(* --- decide -------------------------------------------------------------------
   An end stop is driven into rather than stopped at: the motor keeps running for
   T_EndStop once the estimate reaches the limit, which is what makes the position
   measured there rather than integrated forever, and what lets a cover that has
   drifted find itself again. *)
(* --- a full command re-references, and does not trust the estimate ------------
   The run is timed from the whole travel time rather than from the distance the
   estimate believes is left. That distinction is the difference between a cover
   that heals and one that cannot: if the estimate reads 80 while the shutter is
   at 20, a run of "the remaining 20%" ends nowhere near the stop and the error
   survives. A run of the full travel always ends against it.

   The timer only accumulates while a motor is actually turning, so a fbLockout
   delay or a PRIO_LOCK pause does not eat into the travel - and a lock that
   interrupts a run restarts it from the beginning, which is the safe direction to
   fail in. *)
IF rTarget >= 100.0 THEN
	tRefTime := T_TravelUp + T_EndStop;
ELSE
	tRefTime := T_TravelDown + T_EndStop;
END_IF

fbRefRun(IN := bReferencing AND (iDrivingLast <> ciDriveStop), PT := tRefTime);

IF iManualDrive <> ciDriveStop THEN
	iDriving := iManualDrive;

ELSIF bArrived THEN
	(* Nothing outstanding. Without this the motor restarts the moment a timer
	   resets, and the cover hunts at the limit forever. *)
	iDriving := ciDriveStop;

ELSIF bReferencing THEN
	IF fbRefRun.Q THEN
		(* Against the stop by the clock. This is the one moment the position is
		   measured rather than integrated, so the estimate is set, not nudged. *)
		iDriving := ciDriveStop;
		bArrived := TRUE;
		bReferencing := FALSE;
		PositionKnown := TRUE;
		IF rTarget >= 100.0 THEN
			rPositionReal := 100.0;
		ELSE
			rPositionReal := 0.0;
		END_IF
	ELSIF rTarget >= 100.0 THEN
		iDriving := ciDriveUp;
	ELSE
		iDriving := ciDriveDown;
	END_IF

ELSIF (rTarget - rPositionReal) > BYTE_TO_REAL(Tolerance) THEN
	iDriving := ciDriveUp;

ELSIF (rPositionReal - rTarget) > BYTE_TO_REAL(Tolerance) THEN
	iDriving := ciDriveDown;

ELSE
	(* Close enough. A shutter cannot be positioned finer than its own start and
	   stop time, so this is where a mid-range journey ends - and a mid-range
	   journey is the one case that cannot re-reference, because it does not go
	   anywhere the position is known. *)
	iDriving := ciDriveStop;
	bArrived := TRUE;
END_IF

IF PRIO_LOCK THEN
	iDriving := ciDriveStop;
END_IF

(* --- fbLockout ------------------------------------------------------------------
   A reversing contactor must never be asked to change direction while the motor
   is still turning, so a direction change always passes through a stop of at
   least T_Lockout. Starting from standstill is not delayed. *)
IF (iDriving <> ciDriveStop) AND (iDrivingLast <> ciDriveStop) AND (iDriving <> iDrivingLast) THEN
	iDriving := ciDriveStop;
END_IF

(* The timer runs on where the cover WAS, not on what has just been decided.
   Feeding it the decision deadlocks the block: asking to move makes IN FALSE,
   which resets the very timer that would have permitted moving, so the request
   is refused again on the next cycle and forever after. That cost a bench run,
   and the symptom was a cover that byReported STOPPED at 0% no matter what was
   asked of it. *)
fbLockout(IN := (iDrivingLast = ciDriveStop), PT := T_Lockout);

IF (iDriving <> ciDriveStop) AND (iDrivingLast = ciDriveStop) AND NOT fbLockout.Q THEN
	(* Stopped too recently to start again - the contactor gets its dead time. *)
	iDriving := ciDriveStop;
END_IF

iDrivingLast := iDriving;

MU := (iDriving = ciDriveUp);
MD := (iDriving = ciDriveDown);
Moving := MU OR MD;
Position := REAL_TO_BYTE(rPositionReal + 0.5);

(* --- what to tell Home Assistant ---------------------------------------------
   Position is the estimate, and the estimate is a guess until something has
   driven to an end stop. Publishing that guess as exactly 0 or 100 is worse than
   imprecise: Home Assistant reads those as the limits and disables the button in
   that direction, which is precisely the command that would have re-referenced
   the cover. So an unreferenced cover reports 1 or 99 instead, the slider keeps
   both ends reachable, and one full command puts the matter to rest.

   The Position output is deliberately left alone - logic on the PLC side should
   see the estimate, not a number bent for a user interface. *)
byReported := Position;
IF NOT PositionKnown THEN
	IF byReported >= 100 THEN
		byReported := 99;
	ELSIF byReported = 0 THEN
		byReported := 1;
	END_IF
END_IF

(* --- sState -------------------------------------------------------------------
   Moving beats resting, and an end stop beats the middle. A cover that has not
   reached a stop since power-up says STOPPED rather than guessing: the estimate
   starts at 0, which looks exactly like a shutter resting closed and is in fact
   an assumption. FB_OUTPUT_COVER_MQTT publishes STOPPED at boot for the same
   reason. *)
IF MU THEN
	sState := 'OPENING';
ELSIF MD THEN
	sState := 'CLOSING';
ELSIF NOT PositionKnown THEN
	sState := 'STOPPED';
ELSIF Position >= 100 THEN
	sState := 'OPEN';
ELSIF Position = 0 THEN
	sState := 'CLOSED';
ELSE
	sState := 'STOPPED';
END_IF

IF bInitMqttDone AND (bStartup OR (sState <> sPublishedState)) THEN
	sPublishedState := sState;
	pMqttPublishQueue^.AddMessage(
		Payload := sState,
		Topic := THIS^.sMQTTPublishTopic,
		Qos := MQTT.QoS.ExactlyOnce,
		MqttRetain := TRUE);
END_IF

(* --- position ----------------------------------------------------------------
   While moving, every PublishStep percent, so the slider tracks the shutter
   without flooding the broker. When movement ends, the exact value, because that
   is the number somebody will read off a dashboard for the next hour. *)
IF bInitMqttDone THEN
	iDiff := BYTE_TO_INT(byReported) - BYTE_TO_INT(byPublishedPosition);
	IF iDiff < 0 THEN
		iDiff := -iDiff;
	END_IF

	IF bStartup
		OR NOT bPositionPublished
		OR (NOT Moving AND (byReported <> byPublishedPosition))
		OR (iDiff >= BYTE_TO_INT(PublishStep))
	THEN
		byPublishedPosition := byReported;
		bPositionPublished := TRUE;
		Payload := BYTE_TO_STRING(byReported);
		pMqttPublishQueue^.AddMessage(
			Payload := Payload,
			Topic := PositionTopic,
			Qos := MQTT.QoS.ExactlyOnce,
			MqttRetain := TRUE);
	END_IF

	bStartup := FALSE;
END_IF

          

(* Callback invoked by the callback collector when a message arrives on the subscribed topic. Not called directly. *)
METHOD PublishReceived : BOOL
  VAR_INPUT
    Data : MQTT.CALLBACK_DATA;  (* Collection of recived Data *)
  END_VAR
                  //first check if Mqtt is initialized, otherwise do nothing
IF NOT(bInitMqttDone) THEN
	//mark the interface call from the collector as done
	PublishReceived := TRUE;

//the command topic: the same three payloads the older cover block takes
ELSIF CommonTypesAndFunctions.StrEquals(str1:= ADR(sMQTTSubscribeTopic), str2:= Data.TopicOut) THEN
	PublishReceived := TRUE;
	IF CommonTypesAndFunctions.StrEquals(str1:= Data.PayloadString, str2:= ADR('STOP')) THEN
		THIS^.bMqttRequestStop := TRUE;
	ELSIF CommonTypesAndFunctions.StrEquals(str1:= Data.PayloadString, str2:= ADR('OPEN')) THEN
		THIS^.bMqttRequestOpen := TRUE;
	ELSIF CommonTypesAndFunctions.StrEquals(str1:= Data.PayloadString, str2:= ADR('CLOSE')) THEN
		THIS^.bMqttRequestClose := TRUE;
	END_IF

//and the position topic, which carries a bare number
ELSIF CommonTypesAndFunctions.StrEquals(str1:= ADR(SetPositionTopic), str2:= Data.TopicOut) THEN
	PublishReceived := TRUE;
	(* Home Assistant sends the number as text. STRING_TO_BYTE returns 0 for
	   anything it cannot parse, which is indistinguishable from a genuine
	   request to close - so an unparseable payload is dropped instead, and
	   'closed' has to be asked for as 0 or as CLOSE. *)
	IF CommonTypesAndFunctions.StrEquals(str1:= Data.PayloadString, str2:= ADR('0'))
		OR (STRING_TO_BYTE(Data.PayloadString^) > 0)
	THEN
		THIS^.byMqttRequestPositionPct := STRING_TO_BYTE(Data.PayloadString^);
		IF THIS^.byMqttRequestPositionPct > 100 THEN
			THIS^.byMqttRequestPositionPct := 100;
		END_IF
		THIS^.bMqttRequestPosition := TRUE;
	END_IF
END_IF

                
END_METHOD

(* Publishes the Home Assistant MQTT discovery config so the entity is created automatically, with a position slider. Call once at bStartup, after InitMqtt. *)
METHOD InitMqttDiscovery
  VAR_INPUT
    Device : POINTER TO FB_PLC_MQTT_DISCOVERY_DEVICE;  (* Pointer to the discovery device this entity belongs to, normally GVL_MQTT.PLC_Device. *)
    Name : STRING(255);  (* Name of the entity in Home Assistant. The self-wiring prologue passes FriendlyName. *)
    overruleId : STRING(255) := '';  (* Overrides the generated entity id. Leave empty to derive it from the function block name. *)
    DeviceClass : STRING(50) := 'shutter';  (* Home Assistant cover device class - shutter, blind, awning, curtain, shade, garage, gate. It changes the icon and the words on the buttons, not the behaviour. *)
  END_VAR
  VAR
    id : STRING(255);  (* Resolved entity id. *)
  END_VAR
                  IF bInitMqttDone AND NOT bInitMqttDiscoveryDone THEN

	id := SUPER^.ResolveEntityId(overruleId);

	(* A different method, not extra arguments to the one FB_OUTPUT_COVER_MQTT uses:
	   Home Assistant rejects position_topic and set_position_topic as null, so the
	   two configs have to differ by which keys exist rather than by their values.
	   Everything else is deliberately identical, so swapping one block for the
	   other keeps the same behaviour for open, close and stop. *)
	Device^.CreateCoverEntityWithPosition(
		Name := name,
		Id := id,
		CommandTopic := THIS^.sMQTTSubscribeTopic,
		PayloadOpen := 'OPEN',
		PayloadClose := 'CLOSE',
		PayloadStop := 'STOP',
		StateTopic := THIS^.sMQTTPublishTopic,
		StateOpen := 'OPEN',
		StateOpening := 'OPENING',
		StateClosed := 'CLOSED',
		StateClosing := 'CLOSING',
		StateStopped := 'STOPPED',
		DeviceClass := DeviceClass,
		PositionTopic := CONCAT(THIS^.sMQTTPublishTopic, '/POSITION'),
		SetPositionTopic := CONCAT(THIS^.sMQTTSubscribeTopic, '/POSITION'),
		PositionOpen := 100,
		PositionClosed := 0);

	bInitMqttDiscoveryDone := TRUE;
END_IF
                
END_METHOD

(* Enables MQTT on the function block. Call once at bStartup. Not needed when FriendlyName is set at the declaration: the block then wires itself. *)
METHOD InitMqtt
  VAR_INPUT
    MQTTPublishPrefix : POINTER TO STRING;  (* Pointer to the MQTT publish prefix used for this block. The function block name is appended automatically. *)
    MQTTSubscribePrefix : POINTER TO STRING;  (* Pointer to the MQTT subscribe prefix used for this block. *)
    pMqttPublishQueue : POINTER TO FB_MQTT_PUBLISH_QUEUE;  (* Pointer to the shared MQTT queue that carries messages to the broker. *)
    pMqttCallbackCollector : POINTER TO MQTT.CallbackCollector;  (* Pointer to the callback collector this block registers with, so commands reach it. *)
  END_VAR
                  SUPER^._sInstancePath := THIS^.sInstancePath; // Due to reflection its location is important

(*pass trough*)
THIS^.pMqttPublishQueue := pMqttPublishQueue;
THIS^.psMqttPublishTopicPrefix := MQTTPublishPrefix;
THIS^.psMqttSubscribeTopicPrefix := MQTTSubscribePrefix;

SUPER^.InitBaseMqtt();
pMqttCallbackCollector^.put(instance := THIS^); // register the FB against the collector so mqtt events can be received

                
END_METHOD
END_FUNCTION_BLOCK

{attribute 'reflection'}
FUNCTION_BLOCK FB_OUTPUT_DIMMER_MQTT EXTENDS FB_MQTT_BASE IMPLEMENTS MQTT.MQTT_SUBSCRIBE_CALLBACK
  VAR_OUTPUT
    Q : BOOL;
    Q_OUT : WORD;
    OUT : WORD;
  END_VAR
  VAR
    fbT3 : OSCAT_BASIC.TON;
    dim : OSCAT_BASIC._RMP_B;
    dir : BOOL;
    byOutInternal : BYTE;
    LIN_TRAFO : Util.LIN_TRAFO;
    OUT_LinearScaleMin : INT := 0;
    OUT_LinearScaleMax : INT := 32767;
    {attribute 'noinit'}
    {attribute 'instance-path'}
    sInstancePath : STRING(GVL_MQTT.MQTT_TOPIC_LEN);  (* Refelection: object's full instance name *)
    bStartup : BOOL := TRUE;
    OutputDimmer : BOOL;
    Qos_Dimm : MQTT.QoS;
    Delta_Dimm : INT := 1;  (* Minimum brightness change before republishing. 0 would publish every scan. *)
    T_Debounce : TIME := TIME#10ms;  (* Default values for E_DIMMER, can be overwritten by method call *)
    T_Reconfig : TIME := TIME#10s0ms;
    T_On_Max : TIME := TIME#0ms;
    T_Dimm_Start : TIME := TIME#400ms;
    T_Dimm : TIME := TIME#3s0ms;
    Min_On : BYTE := 50;
    Max_On : BYTE := 255;
    Soft_Dimm : BOOL := TRUE;
    Rst_Out : BOOL := FALSE;
  END_VAR
  VAR PERSISTENT
    byPreviousOUT : BYTE;  (* To retain output state through powercycles *)
    bPreviousQ : BOOL;  (* To retain output state through powercycles *)
  END_VAR
  VAR_INPUT
    SINGLE : BOOL;
    LONG : BOOL;
    P_LONG : BOOL;
    PRIO_HIGH : BOOL := FALSE;
    PRIO_LOW : BOOL := FALSE;
    SET : BOOL;
    VAL : BYTE;
    RST : BOOL;
  END_VAR

            (* --- self-wiring prologue ----------------------------------------------------
   Makes the InitMqtt and InitMqttDiscovery* calls optional. Set FriendlyName at
   the declaration site and this block wires itself from GVL_MQTT on its
   first cyclic call, then announces itself to Home Assistant.

   Deliberately in the body rather than in FB_init: it dereferences GVL members
   and reads the reflection instance path, and doing that during initialisation
   would rely on an ordering nothing enforces and the compiler cannot check. The
   body is the same lifecycle phase the init actions used, so this is not merely
   safe, it is the phase that already works today.

   The wiring calls this block's own unmodified InitMqtt / InitMqttDiscovery*
   methods, so anything published - topics and discovery JSON alike - is produced
   by exactly the code that produces it today. Only the trigger moved.

   Dormant while FriendlyName is empty, so existing projects and existing call
   sites keep working untouched.

   A block wired this way MUST be called cyclically. An instance whose body never
   runs is now unwired and absent from Home Assistant, where the init action used
   to wire it regardless. Nothing warns about that.  *)
IF FriendlyName <> '' THEN

	IF NOT bInitMqttDone THEN
		THIS^.InitMqtt(
			MQTTPublishPrefix := ADR(GVL_MQTT.MqttPubDimmerPrefix),
			MQTTSubscribePrefix := ADR(GVL_MQTT.MqttSubDimmerPrefix),
			pMqttPublishQueue := ADR(GVL_MQTT.fbMqttPublishQueue),
			pMqttCallbackCollector := ADR(GVL_MQTT.collector_FB_DIMMER_MQTT),
			OutputDimmer := TRUE,
			Qos_Dimm := MQTT.QoS.ExactlyOnce,
			Delta_Dimm := 5);
	END_IF

	IF bInitMqttDone AND NOT bInitMqttDiscoveryDone THEN
		THIS^.InitMqttDiscovery(
			Device := ADR(GVL_MQTT.PLC_Device),
			Name := FriendlyName);
	END_IF

END_IF

IF bStartup THEN
	byOutInternal := byPreviousOUT;
	Q := bPreviousQ;
END_IF

IF RST THEN
	IF rst_out THEN byOutInternal := 0; END_IF;
	Q := FALSE;
	dir := byOutInternal > 127;
ELSIF PRIO_HIGH THEN
	Q := TRUE;
	byOutInternal := 255;
ELSIF PRIO_LOW THEN
	Q := FALSE;
ELSIF bMqttHighRequest THEN
	Q:= TRUE;
	bMqttHighRequest := FALSE;
	bMqttLowRequest := FALSE;
ELSIF bMqttLowRequest THEN
	Q:= FALSE;
	bMqttHighRequest := FALSE;
	bMqttLowRequest := FALSE;
ELSIF set THEN
	byOutInternal := val;
	Q := TRUE;
	(* set direction to up when value < 127 otherwise set dir down dir is reversed because next action will reverse again *)
	dir := byOutInternal > 127;
ELSIF SINGLE THEN
	(* a single click reverses output Q *)
	Q := NOT Q;
	(* when E_DIMMER is turned on we need to limit out to min and max limits *)
	IF Q THEN byOutInternal := LIMIT(MAX(byOutInternal,1), byOutInternal, MAX_ON);	END_IF;
	(* set the appropriate direction of E_DIMMER dir is reversed because next action will reverse again *)
	dir := byOutInternal > 127;
ELSIF LONG THEN
	IF NOT Q THEN
		IF SOFT_DIMM THEN
			byOutInternal := 1;
			dir := TRUE;
		ELSE
			byOutInternal := LIMIT(MAX(MIN_ON,1), byOutInternal, MAX_ON);
			DIR := byOutInternal < 127;
		END_IF;
		Q := TRUE;
	ELSE
		(* reverse direction with every long click *)
		dir := NOT dir;
	END_IF;
END_IF;


(* while dimming is active ramp the output out up or down *)
dim(DIR := dir, e := P_LONG AND Q, TR := T_DIMM, rmp := byOutInternal);

(* reverse direction when limits are reached *)
IF byOutInternal = 0 THEN
	dir := TRUE;
ELSIF byOutInternal = 255 THEN
	dir := FALSE;
END_IF;

(* limit the maximum runtime *)
IF t_ON_MAX > t#0s THEN
	fbT3(in := q, pt := T_ON_MAX);
	Q := Q XOR fbT3.Q;
END_IF;

(* Scale the internal OUT to the actual OUT *)
LIN_TRAFO(
		IN:= byOutInternal,
		IN_MIN:= 0,
		IN_MAX:= 255,
		OUT_MIN:=OUT_LinearScaleMin,
		OUT_MAX:=OUT_LinearScaleMax
	);
OUT:= REAL_TO_WORD(LIN_TRAFO.OUT);
IF Q THEN
	Q_OUT:= OUT;
ELSE
	Q_OUT:= 0;
END_IF

IF ((ABS(BYTE_TO_INT(byPreviousOUT) - BYTE_TO_INT(byOutInternal)) >= Delta_Dimm AND byOutInternal <> byPreviousOUT) OR bStartup AND byOutInternal <> byPreviousOUT OR bStartup AND OutputDimmer) AND bInitMqttDone THEN
	byPreviousOUT:=byOutInternal;
	pMqttPublishQueue^.AddMessage(		
		Payload := BYTE_TO_STRING(byOutInternal),
		Topic := CONCAT(CONCAT(psMqttPublishTopicPrefix^, MqttPublishTopicSuffix), '/OUT'),
		Qos := MQTT.QoS.ExactlyOnce,
		MqttRetain := TRUE
	);
END_IF

IF (Q <> bPreviousQ OR bStartup) AND bInitMqttDone THEN
	bPreviousQ:=Q;
	pMqttPublishQueue^.AddMessage(
		Payload := BOOL_TO_STRING(Q),
		Topic := CONCAT(CONCAT(psMqttPublishTopicPrefix^, MqttPublishTopicSuffix), '/Q'),
		Qos := Qos_Dimm,
		MqttRetain := TRUE
	);
END_IF

bStartup:=FALSE;
          

METHOD PublishReceived : BOOL
  VAR_INPUT
    Data : MQTT.CALLBACK_DATA;  (* Collection of recived Data *)
  END_VAR
                  //first check if Mqtt is initialized, otherwise do nothing
IF NOT(bInitMqttDone) THEN
	//mark the interface call from the collector as done
	PublishReceived := TRUE;
//check if the packet is for this FB
ELSIF CONCAT(sMQTTSubscribeTopic,'/Q') =  Data.TopicOut^ THEN
	//mark the interface call from the collector as done
	PublishReceived := TRUE;
	IF CommonTypesAndFunctions.StrEquals(str1:= Data.PayloadString, str2:= ADR('TRUE')) THEN
		bMqttHighRequest := TRUE;
	ELSIF CommonTypesAndFunctions.StrEquals(str1:= Data.PayloadString, str2:= ADR('FALSE')) THEN
		bMqttLowRequest := TRUE;
	END_IF;
	
ELSIF CONCAT(sMQTTSubscribeTopic,'/OUT') =  Data.TopicOut^ THEN
	//mark the interface call from the collector as done
	PublishReceived := TRUE;
	IF OSCAT_BASIC.IS_CC(str:= Data.PayloadString^,cmp:='0123456789.') AND THIS^.PRIO_HIGH = FALSE THEN
		THIS^.byOutInternal:=STRING_TO_BYTE(Data.PayloadString^);
	END_IF
END_IF
                
END_METHOD

METHOD ConfigureFunctionBlock
  VAR_INPUT
    T_Debounce : TIME := TIME#10ms;  (* Default values for E_DIMMER, can be overwritten by method call *)
    T_Reconfig : TIME := TIME#10s0ms;
    T_On_Max : TIME := TIME#0ms;
    T_Dimm_Start : TIME := TIME#400ms;
    T_Dimm : TIME := TIME#3s0ms;
    Min_On : BYTE := 50;
    Max_On : BYTE := 255;
    Soft_Dimm : BOOL := TRUE;
    Rst_Out : BOOL := FALSE;
    OUT_LinearScaleMin : INT := 0;
    OUT_LinearScaleMax : INT := 32767;
  END_VAR
                  THIS^.T_Debounce:=T_Debounce;
THIS^.T_Reconfig:=T_Reconfig;
THIS^.T_On_Max:=T_On_Max;
THIS^.T_Dimm_Start:=T_Dimm_Start;
THIS^.T_Dimm:=T_Dimm;
THIS^.Min_On:=Min_On;
THIS^.Max_On:=Max_On;
THIS^.Soft_Dimm:=Soft_Dimm;
THIS^.Rst_Out:=Rst_Out;
THIS^.OUT_LinearScaleMin:=OUT_LinearScaleMin;
THIS^.OUT_LinearScaleMax:=OUT_LinearScaleMax;
                
END_METHOD

METHOD InitMqtt
  VAR_INPUT
    MQTTPublishPrefix : POINTER TO STRING;
    MQTTSubscribePrefix : POINTER TO STRING;
    pMqttPublishQueue : POINTER TO FB_MQTT_PUBLISH_QUEUE;
    pMqttCallbackCollector : POINTER TO MQTT.CallbackCollector;
    OutputDimmer : BOOL;  (* E_DIMMER specific *)
    Qos_Dimm : MQTT.QoS;
    Delta_Dimm : INT;
  END_VAR
                  SUPER^._sInstancePath := THIS^.sInstancePath; // Due to reflection its location is important

(*pass trough*)
THIS^.pMqttPublishQueue := pMqttPublishQueue;
THIS^.psMqttPublishTopicPrefix:=MQTTPublishPrefix;
THIS^.psMqttSubscribeTopicPrefix:=MQTTSubscribePrefix;
THIS^.pMqttPublishQueue:=pMqttPublishQueue;

// E_DIMMER specific
THIS^.OutputDimmer:=OutputDimmer;
THIS^.Qos_Dimm:=Qos_Dimm;
THIS^.Delta_Dimm:=Delta_Dimm;


SUPER^.InitBaseMqtt();
pMqttCallbackCollector^.put(instance:= THIS^); // register the FB agains the collector so mqtt events can be received


                
END_METHOD

METHOD InitMqttDiscovery
  VAR_INPUT
    Device : POINTER TO FB_PLC_MQTT_DISCOVERY_DEVICE;
    Name : STRING(255);
    overruleId : STRING(255) := '';
  END_VAR
  VAR
    id : STRING(255);
  END_VAR
                  IF bInitMqttDone AND NOT bInitMqttDiscoveryDone THEN
	
	id := SUPER^.ResolveEntityId(overruleId);
	
	Device^.CreateLightDimmerEntity(
		Name := name,
		Id := Id,
		CommandTopic := CONCAT(THIS^.sMQTTSubscribeTopic,'/Q'),
		PayloadOn := 'TRUE',
		PayloadOff := 'FALSE',
		StateTopic := CONCAT(THIS^.sMQTTPublishTopic,'/Q'),
		BrightnessCommandTopic := CONCAT(THIS^.sMQTTSubscribeTopic,'/OUT'),
		BrightnessStateTopic := CONCAT(THIS^.sMQTTPublishTopic,'/OUT'),
		BrightnessScale := 255);

	bInitMqttDiscoveryDone := TRUE;
END_IF
                
END_METHOD
END_FUNCTION_BLOCK

{attribute 'reflection'}
FUNCTION_BLOCK FB_OUTPUT_DIMMER_DALI_MQTT EXTENDS FB_MQTT_BASE IMPLEMENTS MQTT.MQTT_SUBSCRIBE_CALLBACK
  VAR_OUTPUT
    STATUS_LED : BOOL;
  END_VAR
  VAR
    {attribute 'noinit'}
    {attribute 'instance-path'}
    sInstancePath : STRING(GVL_MQTT.MQTT_TOPIC_LEN);  (* Refelection: object's full instance name *)
    bStartup : BOOL := TRUE;
    fbDaliSendDimValue : WagoAppDALI.FbDaliSendDimValue;
    fbDaliSendFadeTime : WagoAppDALI.FbDaliSendFadeTime;
    fbDaliSendFadeRate : WagoAppDALI.FbDaliSendFadeRate;
    bMqttSendBrightnessUpdate : BOOL;
    bMqttSendOnUpdate : BOOL;
    bMqttSendOffUpdate : BOOL;
    fbToggleRTrigger : Standard.R_TRIG;
    fbDaliSyncSignalGenerator : Util.BLINK;
    fbDaliConfigSyncSignalGenerator : Util.BLINK;
    iDimDirection : INT := 1;
  END_VAR
  VAR PERSISTENT
    rDimValue : REAL;
  END_VAR
  VAR_INPUT
    BALLAST : WagoAppDALI.typBallast;
    TOGGLE : BOOL;
    P_LONG : BOOL;
    PRIO_HIGH : BOOL := FALSE;
    PRIO_LOW : BOOL := FALSE;
  END_VAR

            fbDaliSendFadeTime(
	typBallast := BALLAST,
	bFadeTime := 2, // 1 sec
	xUpdate := fbDaliConfigSyncSignalGenerator.OUT
	);
	
fbDaliSendFadeRate(
	typBallast := BALLAST,
	bFadeRate := 2, // 1 sec
	xUpdate := fbDaliConfigSyncSignalGenerator.OUT
	);

fbDaliSendDimValue(
	typBallast := BALLAST,
	rDimValue := rDimValue,
	xUpdate := fbDaliSyncSignalGenerator.OUT OR bMqttSendOffUpdate OR bMqttSendOnUpdate);

fbDaliSyncSignalGenerator(
	ENABLE := TRUE,
	TIMEHIGH := T#1S,
	TIMELOW := T#1M);
	
fbDaliConfigSyncSignalGenerator(
	ENABLE := TRUE,
	TIMEHIGH := T#1S,
	TIMELOW := T#24H);

fbToggleRTrigger(CLK:=TOGGLE);

// Regular push
IF(fbToggleRTrigger.Q AND rDimValue = 0) THEN
	SetDimValue(100);
ELSIF(fbToggleRTrigger.Q AND rDimValue > 0) THEN
	SetDimValue(0);
END_IF

// Long push
IF P_LONG THEN
	SetDimValue(rDimValue + iDimDirection);
END_IF

IF bMqttSendBrightnessUpdate OR bStartup AND bInitMqttDone THEN
	pMqttPublishQueue^.AddMessage(		
		Payload := REAL_TO_STRING(rDimValue),
		Topic := CONCAT(THIS^.sMQTTPublishTopic, '/BRIGHTNESS'),
		Qos := MQTT.QoS.ExactlyOnce,
		MqttRetain := TRUE
	);
	bMqttSendBrightnessUpdate := FALSE;
END_IF

IF bMqttSendOnUpdate OR (bStartup AND rDimValue > 0) AND bInitMqttDone THEN
	pMqttPublishQueue^.AddMessage(		
		Payload := 'ON',
		Topic := THIS^.sMQTTPublishTopic,
		Qos := MQTT.QoS.ExactlyOnce,
		MqttRetain := TRUE
	);
	bMqttSendOnUpdate := FALSE;
END_IF

IF bMqttSendOffUpdate OR (bStartup AND rDimValue = 0) AND bInitMqttDone THEN
	pMqttPublishQueue^.AddMessage(
		Payload := 'OFF',
		Topic := THIS^.sMQTTPublishTopic,
		Qos := MQTT.QoS.ExactlyOnce,
		MqttRetain := TRUE
	);
	bMqttSendOffUpdate := FALSE;
END_IF

bStartup:=FALSE;
STATUS_LED := REAL_TO_BOOL(rDimValue);
          

METHOD InitMqttDiscovery
  VAR_INPUT
    Device : POINTER TO FB_PLC_MQTT_DISCOVERY_DEVICE;
    Name : STRING(255);
    overruleId : STRING(255) := '';
  END_VAR
  VAR
    id : STRING(255);
  END_VAR
                  IF bInitMqttDone AND NOT bInitMqttDiscoveryDone THEN
	
	IF CommonTypesAndFunctions.StrEquals(str1:= ADR(overruleId), str2:= ADR('')) THEN
		id := CONCAT(CONCAT(THIS^.DeviceName,'_'), THIS^.psInstanceNamePt^); // 'FB_DI_PB_003'
	ELSE
		id := overruleId; // 'MY_PH_GND_HALL_01'
	END_IF
	
	Device^.CreateLightDimmerEntity(
		Name := name,
		Id := Id,
		CommandTopic := THIS^.sMQTTSubscribeTopic,
		PayloadOn := 'ON',
		PayloadOff := 'OFF',
		StateTopic := THIS^.sMQTTPublishTopic,
		BrightnessCommandTopic := CONCAT(THIS^.sMQTTSubscribeTopic, '/BRIGHTNESS'),
		BrightnessStateTopic := CONCAT(THIS^.sMQTTPublishTopic, '/BRIGHTNESS'),
		BrightnessScale := 100,
		OnCommandType := 'brightness');

	bInitMqttDiscoveryDone := TRUE;
END_IF
                
END_METHOD

METHOD InitMqtt
  VAR_INPUT
    MQTTPublishPrefix : POINTER TO STRING;
    MQTTSubscribePrefix : POINTER TO STRING;
    pMqttPublishQueue : POINTER TO FB_MQTT_PUBLISH_QUEUE;
    pMqttCallbackCollector : POINTER TO MQTT.CallbackCollector;
  END_VAR
                  SUPER^._sInstancePath := THIS^.sInstancePath; // Due to reflection its location is important

(*pass trough*)
THIS^.pMqttPublishQueue := pMqttPublishQueue;
THIS^.psMqttPublishTopicPrefix:=MQTTPublishPrefix;
THIS^.psMqttSubscribeTopicPrefix:=MQTTSubscribePrefix;
THIS^.pMqttPublishQueue:=pMqttPublishQueue;

SUPER^.InitBaseMqtt();
pMqttCallbackCollector^.put(instance:= THIS^); // register the FB agains the collector so mqtt events can be received


                
END_METHOD

METHOD PublishReceived : BOOL
  VAR_INPUT
    Data : MQTT.CALLBACK_DATA;  (* Collection of recived Data *)
  END_VAR
                  //first check if Mqtt is initialized, otherwise do nothing
IF NOT(bInitMqttDone) THEN
	//mark the interface call from the collector as done
	PublishReceived := TRUE;
	
ELSIF sMQTTSubscribeTopic =  Data.TopicOut^ THEN
	IF CommonTypesAndFunctions.StrEquals(str1:= Data.PayloadString, str2:= ADR('ON')) THEN
		SetDimValue(100);
	ELSIF CommonTypesAndFunctions.StrEquals(str1:= Data.PayloadString, str2:= ADR('OFF')) THEN
		SetDimValue(0);
	END_IF
	
ELSIF CONCAT(sMQTTSubscribeTopic, '/BRIGHTNESS') =  Data.TopicOut^ THEN
	IF OSCAT_BASIC.IS_CC(str:= Data.PayloadString^,cmp:='0123456789.') AND THIS^.PRIO_HIGH = FALSE THEN
		SetDimValue(STRING_TO_REAL(Data.PayloadString^));
	END_IF
END_IF 
                
END_METHOD

METHOD SetDimValue
  VAR_INPUT
    Value : REAL;
  END_VAR
                  THIS^.bMqttSendBrightnessUpdate := TRUE;

IF THIS^.rDimValue = 0 AND Value > 0 THEN
	THIS^.bMqttSendOnUpdate := TRUE;
END_IF

IF THIS^.rDimValue > 0 AND Value = 0 THEN
	THIS^.bMqttSendOffUpdate := TRUE;
END_IF

IF Value = 0 THEN
	iDimDirection := 1;
ELSIF Value = 100 THEN
	iDimDirection := -1;
END_IF

THIS^.rDimValue := Value;
                
END_METHOD

METHOD ConfigureFunctionBlock : BOOL
  VAR_INPUT
    FadeTime : BYTE;
    FadeRate : BYTE;
  END_VAR
                  fbDaliSendFadeTime.bFadeTime := FadeTime;
fbDaliSendFadeRate.bFadeRate := FadeRate;
                
END_METHOD
END_FUNCTION_BLOCK

{attribute 'reflection'}
FUNCTION_BLOCK FB_OUTPUT_DIMMER_DMX_MQTT EXTENDS FB_MQTT_BASE IMPLEMENTS MQTT.MQTT_SUBSCRIBE_CALLBACK
  VAR_OUTPUT
    Q : BOOL;
    Q_OUT : WORD;
    OUT : WORD;
  END_VAR
  VAR
    {attribute 'noinit'}
    {attribute 'instance-path'}
    sInstancePath : STRING(GVL_MQTT.MQTT_TOPIC_LEN);  (* Refelection: object's full instance name *)
    fbT3 : OSCAT_BASIC.TON;
    dim : OSCAT_BASIC._RMP_B;
    dir : BOOL;
    byOutInternal : BYTE;
    LIN_TRAFO : Util.LIN_TRAFO;
    bStartup : BOOL := TRUE;
    OutputDimmer : BOOL;
    Qos_Dimm : MQTT.QoS;
    Delta_Dimm : INT := 1;  (* Minimum brightness change before republishing. 0 would publish every scan. *)
    T_Debounce : TIME := TIME#10ms;  (* Default values for E_DIMMER, can be overwritten by method call *)
    T_Reconfig : TIME := TIME#10s0ms;
    T_On_Max : TIME := TIME#0ms;
    T_Dimm_Start : TIME := TIME#400ms;
    T_Dimm : TIME := TIME#1s0ms;
    Min_On : BYTE := 100;
    Max_On : BYTE := 200;
    Soft_Dimm : BOOL := TRUE;
    Rst_Out : BOOL := FALSE;
    OUT_LinearScaleMin : INT := 10000;
    OUT_LinearScaleMax : INT := 32767;
    DmxChannel : INT;  (* DMX specific *)
    DmxWidth : INT;
    DmxUniverse : INT;
    pDmxValues : POINTER TO oscat_network.NETWORK_BUFFER_SHORT;
    bInitDmxDone : BOOL := FALSE;
  END_VAR
  VAR PERSISTENT
    byPreviousOUT : BYTE;  (* To retain output state through powercycles *)
    bPreviousQ : BOOL;  (* To retain output state through powercycles *)
  END_VAR
  VAR_INPUT
    SINGLE : BOOL;
    LONG : BOOL;
    P_LONG : BOOL;
    PRIO_HIGH : BOOL := FALSE;
    PRIO_LOW : BOOL := FALSE;
    SET : BOOL;
    VAL : BYTE;
    RST : BOOL;
  END_VAR

            (* --- self-wiring prologue ----------------------------------------------------
   Makes the InitMqtt and InitMqttDiscovery* calls optional. Set FriendlyName at
   the declaration site and this block wires itself from GVL_MQTT on its
   first cyclic call, then announces itself to Home Assistant.

   Deliberately in the body rather than in FB_init: it dereferences GVL members
   and reads the reflection instance path, and doing that during initialisation
   would rely on an ordering nothing enforces and the compiler cannot check. The
   body is the same lifecycle phase the init actions used, so this is not merely
   safe, it is the phase that already works today.

   The wiring calls this block's own unmodified InitMqtt / InitMqttDiscovery*
   methods, so anything published - topics and discovery JSON alike - is produced
   by exactly the code that produces it today. Only the trigger moved.

   Dormant while FriendlyName is empty, so existing projects and existing call
   sites keep working untouched.

   A block wired this way MUST be called cyclically. An instance whose body never
   runs is now unwired and absent from Home Assistant, where the init action used
   to wire it regardless. Nothing warns about that.  *)
IF FriendlyName <> '' THEN

	IF NOT bInitMqttDone THEN
		THIS^.InitMqtt(
			MQTTPublishPrefix := ADR(GVL_MQTT.MqttPubDimmerPrefix),
			MQTTSubscribePrefix := ADR(GVL_MQTT.MqttSubDimmerPrefix),
			pMqttPublishQueue := ADR(GVL_MQTT.fbMqttPublishQueue),
			pMqttCallbackCollector := ADR(GVL_MQTT.collector_FB_DIMMER_MQTT),
			OutputDimmer := TRUE,
			Qos_Dimm := MQTT.QoS.ExactlyOnce,
			Delta_Dimm := 5);
	END_IF

	IF bInitMqttDone AND NOT bInitMqttDiscoveryDone THEN
		THIS^.InitMqttDiscovery(
			Device := ADR(GVL_MQTT.PLC_Device),
			Name := FriendlyName);
	END_IF

END_IF

IF bStartup THEN
	byOutInternal := byPreviousOUT;
	Q := bPreviousQ;
END_IF

IF RST THEN
	IF rst_out THEN byOutInternal := 0; END_IF;
	Q := FALSE;
	dir := byOutInternal > 127;
ELSIF PRIO_HIGH THEN
	Q := TRUE;
	byOutInternal := 255;
ELSIF PRIO_LOW THEN
	Q := FALSE;
ELSIF bMqttHighRequest THEN
	Q:= TRUE;
	bMqttHighRequest := FALSE;
	bMqttLowRequest := FALSE;
ELSIF bMqttLowRequest THEN
	Q:= FALSE;
	bMqttHighRequest := FALSE;
	bMqttLowRequest := FALSE;
ELSIF set THEN
	byOutInternal := val;
	Q := TRUE;
	(* set direction to up when value < 127 otherwise set dir down dir is reversed because next action will reverse again *)
	dir := byOutInternal > 127;
ELSIF SINGLE THEN
	(* a single click reverses output Q *)
	Q := NOT Q;
	(* when E_DIMMER is turned on we need to limit out to min and max limits *)
	IF Q THEN byOutInternal := LIMIT(MAX(byOutInternal,1), byOutInternal, MAX_ON);	END_IF;
	(* set the appropriate direction of E_DIMMER dir is reversed because next action will reverse again *)
	dir := byOutInternal > 127;
ELSIF LONG THEN
	IF NOT Q THEN
		IF SOFT_DIMM THEN
			byOutInternal := 1;
			dir := TRUE;
		ELSE
			byOutInternal := LIMIT(MAX(MIN_ON,1), byOutInternal, MAX_ON);
			DIR := byOutInternal < 127;
		END_IF;
		Q := TRUE;
	ELSE
		(* reverse direction with every long click *)
		dir := NOT dir;
	END_IF;
END_IF;


(* while dimming is active ramp the output out up or down *)
dim(DIR := dir, e := P_LONG AND Q, TR := T_DIMM, rmp := byOutInternal);

(* reverse direction when limits are reached *)
IF byOutInternal = 0 THEN
	dir := TRUE;
ELSIF byOutInternal = 255 THEN
	dir := FALSE;
END_IF;

(* limit the maximum runtime *)
IF t_ON_MAX > t#0s THEN
	fbT3(in := q, pt := T_ON_MAX);
	Q := Q XOR fbT3.Q;
END_IF;

(* Scale the internal OUT to the actual OUT *)
LIN_TRAFO(
		IN:= byOutInternal,
		IN_MIN:= 0,
		IN_MAX:= 255,
		OUT_MIN:=OUT_LinearScaleMin,
		OUT_MAX:=OUT_LinearScaleMax
	);
OUT:= REAL_TO_WORD(LIN_TRAFO.OUT);
IF Q THEN
	Q_OUT:= OUT;
ELSE
	Q_OUT:= 0;
END_IF

IF ((ABS(BYTE_TO_INT(byPreviousOUT) - BYTE_TO_INT(byOutInternal)) >= Delta_Dimm AND byOutInternal <> byPreviousOUT) OR bStartup AND byOutInternal <> byPreviousOUT OR bStartup AND OutputDimmer) AND bInitMqttDone THEN
	byPreviousOUT:=byOutInternal;
	pMqttPublishQueue^.AddMessage(		
		Payload := BYTE_TO_STRING(byOutInternal),
		Topic := CONCAT(THIS^.sMQTTPublishTopic,'/OUT'),
		Qos := MQTT.QoS.ExactlyOnce,
		MqttRetain := TRUE
	);
END_IF

IF (Q <> bPreviousQ OR bStartup) AND bInitMqttDone THEN
	bPreviousQ:=Q;
	pMqttPublishQueue^.AddMessage(
		Payload := BOOL_TO_STRING(Q),
		Topic := CONCAT(THIS^.sMQTTPublishTopic,'/Q'),
		Qos := Qos_Dimm,
		MqttRetain := TRUE
	);
END_IF

bStartup:=FALSE;

(* DMX specific *)
IF bInitDmxDone THEN 
	IF Q THEN
		IF pDmxValues^.BUFFER[DmxChannel-1] <> byOutInternal THEN
			pDmxValues^.BUFFER[DmxChannel-1] := byOutInternal;
		END_IF
	ELSE 
		IF pDmxValues^.BUFFER[DmxChannel-1] <> 0 THEN
			pDmxValues^.BUFFER[DmxChannel-1] := 0;
		END_IF
	END_IF
END_IF
          

METHOD InitMqttDiscovery
  VAR_INPUT
    Device : POINTER TO FB_PLC_MQTT_DISCOVERY_DEVICE;
    Name : STRING(255);
    overruleId : STRING(255) := '';
  END_VAR
  VAR
    id : STRING(255);
  END_VAR
                  IF bInitMqttDone AND NOT bInitMqttDiscoveryDone THEN
	
	id := SUPER^.ResolveEntityId(overruleId);
	
	Device^.CreateLightDimmerEntity(
		Name := name,
		Id := Id,
		CommandTopic := CONCAT(THIS^.sMQTTSubscribeTopic,'/Q'),
		PayloadOn := 'TRUE',
		PayloadOff := 'FALSE',
		StateTopic := CONCAT(THIS^.sMQTTPublishTopic,'/Q'),
		BrightnessCommandTopic := CONCAT(THIS^.sMQTTSubscribeTopic,'/OUT'),
		BrightnessStateTopic := CONCAT(THIS^.sMQTTPublishTopic,'/OUT'),
		BrightnessScale := 255,
		DmxChannel := THIS^.DmxChannel,
		DmxWidth := THIS^.DmxWidth,
		DmxUniverse := THIS^.DmxUniverse);

	bInitMqttDiscoveryDone := TRUE;
END_IF
                
END_METHOD

METHOD initDMX
  VAR_INPUT
    DmxChannel : INT;
    DmxWidth : INT := 1;
    DmxUniverse : INT := 1;
    pDmxValues : POINTER TO oscat_network.NETWORK_BUFFER_SHORT;
  END_VAR
                  
(* A channel outside 1..512 has no slot in the universe, and DmxChannel - 1 is
   what indexes the buffer - so 0 would write BUFFER[-1]. Refusing to init is
   the only report available here: the method returns nothing and the block
   then stays dormant rather than corrupting whatever precedes the buffer. *)
IF DmxChannel < 1 OR DmxChannel > 512 THEN
	RETURN;
END_IF

IF NOT THIS^.bInitDmxDone THEN
	THIS^.DmxChannel := DmxChannel;
	THIS^.pDmxValues := pDmxValues;
	THIS^.DmxWidth := DmxWidth;
	THIS^.DmxUniverse := DmxUniverse;
	THIS^.bInitDmxDone := TRUE;
END_IF
                
END_METHOD

METHOD InitMqtt
  VAR_INPUT
    MQTTPublishPrefix : POINTER TO STRING;
    MQTTSubscribePrefix : POINTER TO STRING;
    pMqttPublishQueue : POINTER TO FB_MQTT_PUBLISH_QUEUE;
    pMqttCallbackCollector : POINTER TO MQTT.CallbackCollector;
    OutputDimmer : BOOL;  (* E_DIMMER specific *)
    Qos_Dimm : MQTT.QoS;
    Delta_Dimm : INT;
  END_VAR
                  SUPER^._sInstancePath := THIS^.sInstancePath; // Due to reflection its location is important

(*pass trough*)
THIS^.pMqttPublishQueue := pMqttPublishQueue;
THIS^.psMqttPublishTopicPrefix:=MQTTPublishPrefix;
THIS^.psMqttSubscribeTopicPrefix:=MQTTSubscribePrefix;
THIS^.pMqttPublishQueue:=pMqttPublishQueue;

// E_DIMMER specific
THIS^.OutputDimmer:=OutputDimmer;
THIS^.Qos_Dimm:=Qos_Dimm;
THIS^.Delta_Dimm:=Delta_Dimm;


SUPER^.InitBaseMqtt();
pMqttCallbackCollector^.put(instance:= THIS^); // register the FB agains the collector so mqtt events can be received


                
END_METHOD

METHOD ConfigureFunctionBlock
  VAR_INPUT
    T_Debounce : TIME := TIME#10ms;  (* Default values for E_DIMMER, can be overwritten by method call *)
    T_Reconfig : TIME := TIME#10s0ms;
    T_On_Max : TIME := TIME#0ms;
    T_Dimm_Start : TIME := TIME#400ms;
    T_Dimm : TIME := TIME#3s0ms;
    Min_On : BYTE := 50;
    Max_On : BYTE := 255;
    Soft_Dimm : BOOL := TRUE;
    Rst_Out : BOOL := FALSE;
    OUT_LinearScaleMin : INT := 0;
    OUT_LinearScaleMax : INT := 32767;
  END_VAR
                  THIS^.T_Debounce:=T_Debounce;
THIS^.T_Reconfig:=T_Reconfig;
THIS^.T_On_Max:=T_On_Max;
THIS^.T_Dimm_Start:=T_Dimm_Start;
THIS^.T_Dimm:=T_Dimm;
THIS^.Min_On:=Min_On;
THIS^.Max_On:=Max_On;
THIS^.Soft_Dimm:=Soft_Dimm;
THIS^.Rst_Out:=Rst_Out;
THIS^.OUT_LinearScaleMin:=OUT_LinearScaleMin;
THIS^.OUT_LinearScaleMax:=OUT_LinearScaleMax;
                
END_METHOD

METHOD PublishReceived : BOOL
  VAR_INPUT
    Data : MQTT.CALLBACK_DATA;  (* Collection of recived Data *)
  END_VAR
                  //first check if Mqtt is initialized, otherwise do nothing
IF NOT(bInitMqttDone) THEN
	//mark the interface call from the collector as done
	PublishReceived := TRUE;
//check if the packet is for this FB
ELSIF CONCAT(sMQTTSubscribeTopic,'/Q') =  Data.TopicOut^ THEN
	IF CommonTypesAndFunctions.StrEquals(str1:= Data.PayloadString, str2:= ADR('TRUE')) THEN
		bMqttHighRequest := TRUE;
	ELSIF CommonTypesAndFunctions.StrEquals(str1:= Data.PayloadString, str2:= ADR('FALSE')) THEN
		bMqttLowRequest := TRUE;
	END_IF;
	
ELSIF CONCAT(sMQTTSubscribeTopic,'/OUT') =  Data.TopicOut^ THEN
	IF OSCAT_BASIC.IS_CC(str:= Data.PayloadString^,cmp:='0123456789.') AND THIS^.PRIO_HIGH = FALSE THEN
		THIS^.byOutInternal:=STRING_TO_BYTE(Data.PayloadString^);
	END_IF
	
	
// Legacy! backwards compatiably with /+ topics instead of /#
ELSIF CommonTypesAndFunctions.StrEqualsAtStart(str1:= ADR(sMQTTSubscribeTopic), str2:= Data.TopicOut) THEN
	//mark the interface call from the collector as done
	PublishReceived := TRUE;
	//now process the data
	IF CommonTypesAndFunctions.StrEquals(str1:= Data.PayloadString, str2:= ADR('TRUE')) THEN
		bMqttHighRequest := TRUE;
	ELSIF CommonTypesAndFunctions.StrEquals(str1:= Data.PayloadString, str2:= ADR('FALSE')) THEN
		bMqttLowRequest := TRUE;
	ELSIF OSCAT_BASIC.IS_CC(str:= Data.PayloadString^,cmp:='0123456789.') AND THIS^.PRIO_HIGH = FALSE THEN
		THIS^.byOutInternal:=STRING_TO_BYTE(Data.PayloadString^);
	END_IF
END_IF 
                
END_METHOD
END_FUNCTION_BLOCK

FUNCTION F_DUCO_NODE_TYPE : E_RS485_DUCO_NODE_TYPE
  VAR_INPUT
    wRaw : WORD;  (* Read parameter 0 of a node, exactly as the bus returned it. *)
  END_VAR

            (* Module type as reported by read parameter 0, mapped onto the enumeration.

   A CASE rather than a cast, deliberately. The bus can return anything - a Duco
   range that grows a type this project has never seen, or a garbled frame that
   passed CRC - and a cast would hand that straight to code which then indexes a
   register table by it. Everything unrecognised becomes Unknown, and a node in
   that state publishes its raw registers and announces nothing. *)
CASE wRaw OF
	10:		F_DUCO_NODE_TYPE := E_RS485_DUCO_NODE_TYPE.DucoBoxFocus;
	11:		F_DUCO_NODE_TYPE := E_RS485_DUCO_NODE_TYPE.ValveSensorless;
	12:		F_DUCO_NODE_TYPE := E_RS485_DUCO_NODE_TYPE.ValveCO2;
	13:		F_DUCO_NODE_TYPE := E_RS485_DUCO_NODE_TYPE.ValveHumidity;
	14:		F_DUCO_NODE_TYPE := E_RS485_DUCO_NODE_TYPE.UserControl;
	15:		F_DUCO_NODE_TYPE := E_RS485_DUCO_NODE_TYPE.SensorCO2;
	16:		F_DUCO_NODE_TYPE := E_RS485_DUCO_NODE_TYPE.SensorHumidity;
	17:		F_DUCO_NODE_TYPE := E_RS485_DUCO_NODE_TYPE.WindowVentilator;
	18:		F_DUCO_NODE_TYPE := E_RS485_DUCO_NODE_TYPE.SwitchSensor;
	19:		F_DUCO_NODE_TYPE := E_RS485_DUCO_NODE_TYPE.ActuatorBoard;
	24:		F_DUCO_NODE_TYPE := E_RS485_DUCO_NODE_TYPE.ValveHumidityCO2;
ELSE
	F_DUCO_NODE_TYPE := E_RS485_DUCO_NODE_TYPE.Unknown;
END_CASE
          
END_FUNCTION

FUNCTION F_DUCO_SCALED_TEXT : STRING(16)
  VAR_INPUT
    iRaw : INT;  (* The register as a signed integer. Signed because outdoor temperature is a real register on this bus and it goes below zero. *)
    iScale : INT;  (* 10 for temperature, 100 for relative humidity. Duco scales those two differently and nothing else on this bus is scaled at all. *)
  END_VAR
  VAR
    iWhole : INT;
    iFrac : INT;
    sOut : STRING(16);
  END_VAR

            (* Formatted from the integer rather than through REAL_TO_STRING, for the reason
   FB_INPUT_TEMPERATURE_RTD_MQTT gives: REAL_TO_STRING on this runtime produces
   a representation nobody wants on a topic. The register is already a fixed-point
   integer, so dividing it into whole and fraction is both exact and shorter. *)
IF iScale <= 0 THEN
	F_DUCO_SCALED_TEXT := INT_TO_STRING(iRaw);
	RETURN;
END_IF

iWhole	:= iRaw / iScale;
iFrac	:= ABS(iRaw MOD iScale);

sOut := INT_TO_STRING(iWhole);

(* IEC division truncates toward zero, so -5/10 is 0 and the sign is lost on
   everything between -1 and 0. Put it back, or -0.5 C publishes as 0.5. *)
IF iRaw < 0 AND iWhole = 0 THEN
	sOut := CONCAT('-', sOut);
END_IF

sOut := CONCAT(sOut, '.');

(* A hundredths scale needs the leading zero: 4907 is 49.07, not 49.7. *)
IF iScale = 100 AND iFrac < 10 THEN
	sOut := CONCAT(sOut, '0');
END_IF

F_DUCO_SCALED_TEXT := CONCAT(sOut, INT_TO_STRING(iFrac));
          
END_FUNCTION

FUNCTION F_DUCO_STATUS_TEXT : STRING(24)
  VAR_INPUT
    wRaw : WORD;  (* Read parameter 1 of a node, the ventilation status. *)
  END_VAR

            (* The status enumeration from L8000009, resolved to text here rather than in a
   Home Assistant template. The PLC is the only place that knows this mapping is
   fixed, and a template is a second copy of it that goes stale silently.

   Not to be confused with the ACTION parameter, holding 9, which encodes the
   same ideas with different numbers: the action that produces "Manual low" is 2,
   and the status that reports it is 4. F_DUCO_ACTION_TEXT is the other one. *)
CASE wRaw OF
	0:		F_DUCO_STATUS_TEXT := 'Auto';
	1:		F_DUCO_STATUS_TEXT := '10 minutes high';
	2:		F_DUCO_STATUS_TEXT := '20 minutes high';
	3:		F_DUCO_STATUS_TEXT := '30 minutes high';
	4:		F_DUCO_STATUS_TEXT := 'Manual low';
	5:		F_DUCO_STATUS_TEXT := 'Manual medium';
	6:		F_DUCO_STATUS_TEXT := 'Manual high';
	7:		F_DUCO_STATUS_TEXT := 'Unoccupied';
	99:		F_DUCO_STATUS_TEXT := 'Error';
ELSE
	(* Published rather than swallowed: an undocumented status is exactly the
	   thing somebody will need to see when a new component misbehaves. *)
	F_DUCO_STATUS_TEXT := CONCAT('Unknown ', WORD_TO_STRING(wRaw));
END_CASE
          
END_FUNCTION

FUNCTION F_DUCO_TYPE_TEXT : STRING(28)
  VAR_INPUT
    eType : E_RS485_DUCO_NODE_TYPE;
  END_VAR

            (* What a node is, in words, for the diagnostic topic. Home Assistant shows this
   on the node's device page, which is where somebody looks after re-pairing the
   network and wondering which valve moved. *)
CASE eType OF
	E_RS485_DUCO_NODE_TYPE.DucoBoxFocus:		F_DUCO_TYPE_TEXT := 'DucoBox Focus';
	E_RS485_DUCO_NODE_TYPE.ValveSensorless:		F_DUCO_TYPE_TEXT := 'Valve';
	E_RS485_DUCO_NODE_TYPE.ValveCO2:			F_DUCO_TYPE_TEXT := 'CO2 valve';
	E_RS485_DUCO_NODE_TYPE.ValveHumidity:		F_DUCO_TYPE_TEXT := 'Humidity valve';
	E_RS485_DUCO_NODE_TYPE.ValveHumidityCO2:	F_DUCO_TYPE_TEXT := 'Humidity + CO2 valve';
	E_RS485_DUCO_NODE_TYPE.UserControl:			F_DUCO_TYPE_TEXT := 'User control';
	E_RS485_DUCO_NODE_TYPE.SensorCO2:			F_DUCO_TYPE_TEXT := 'CO2 sensor';
	E_RS485_DUCO_NODE_TYPE.SensorHumidity:		F_DUCO_TYPE_TEXT := 'Humidity sensor';
	E_RS485_DUCO_NODE_TYPE.WindowVentilator:	F_DUCO_TYPE_TEXT := 'Window ventilator';
	E_RS485_DUCO_NODE_TYPE.SwitchSensor:		F_DUCO_TYPE_TEXT := 'Switch sensor';
	E_RS485_DUCO_NODE_TYPE.ActuatorBoard:		F_DUCO_TYPE_TEXT := 'Actuator board';
ELSE
	F_DUCO_TYPE_TEXT := 'Unknown';
END_CASE
          
END_FUNCTION

FUNCTION F_JSON_RENAME_KEY : BOOL
  VAR_INPUT
    pJson : POINTER TO BYTE;  (* The composed config, edited in place. *)
    uiSize : UDINT;  (* Capacity of the buffer, so the scan cannot run off the end of it. *)
    sFrom : STRING(32);  (* The quoted key as composed, e.g. '"min_val"'. *)
    sTo : STRING(32);  (* The quoted key to publish, e.g. '"min"'. Must not be longer than sFrom. *)
  END_VAR
  VAR
    pFrom : POINTER TO BYTE;
    pTo : POINTER TO BYTE;
    diLen : DINT;
    diFrom : DINT;
    diTo : DINT;
    diI : DINT;
    diJ : DINT;
    diHit : DINT;
    bMatch : BOOL;
  END_VAR

            (* Rename one key in a composed discovery config, in place.

   This exists because a few Home Assistant keys are IEC operators. A number
   entity needs "min" and "max"; ST will not accept members with those names, and
   PRO_JSON takes the key from the member name - there is no name field on
   JSONVAR to override it. So the struct declares min_val / max_val and the key
   is corrected here, on the way out.

   Byte-wise on purpose. FIND and REPLACE are declared over STRING(255) and this
   buffer is STRING(1500), so calling them would silently narrow the config to
   its first 255 bytes - the same trap that once stopped this PLC publishing any
   discovery at all. Never reach for a string function on this buffer. *)
F_JSON_RENAME_KEY := FALSE;

IF pJson = 0 THEN
	RETURN;
END_IF

pFrom := ADR(sFrom);
pTo := ADR(sTo);

(* Walk to the terminator rather than asking a string function for a length. *)
diFrom := 0;
WHILE (diFrom < 32) AND (pFrom[diFrom] <> 0) DO
	diFrom := diFrom + 1;
END_WHILE
diTo := 0;
WHILE (diTo < 32) AND (pTo[diTo] <> 0) DO
	diTo := diTo + 1;
END_WHILE

(* Shortening only. A longer replacement would have to grow the config, and a
   silent overflow here publishes truncated JSON, which Home Assistant discards
   whole. Refusing is the safe answer. *)
IF (diFrom = 0) OR (diTo = 0) OR (diTo > diFrom) THEN
	RETURN;
END_IF

diLen := 0;
WHILE (diLen < UDINT_TO_DINT(uiSize) - 1) AND (pJson[diLen] <> 0) DO
	diLen := diLen + 1;
END_WHILE

diHit := -1;
FOR diI := 0 TO diLen - diFrom DO
	bMatch := TRUE;
	FOR diJ := 0 TO diFrom - 1 DO
		IF pJson[diI + diJ] <> pFrom[diJ] THEN
			bMatch := FALSE;
			EXIT;
		END_IF
	END_FOR
	IF bMatch THEN
		diHit := diI;
		EXIT;
	END_IF
END_FOR

IF diHit < 0 THEN
	RETURN;
END_IF

(* Overwrite the key, then pull the tail left over the slack, terminator and
   all. Keys are unique in one config, so one pass is the whole job. *)
FOR diJ := 0 TO diTo - 1 DO
	pJson[diHit + diJ] := pTo[diJ];
END_FOR

FOR diJ := diHit + diFrom TO diLen DO
	pJson[diJ - (diFrom - diTo)] := pJson[diJ];
END_FOR

F_JSON_RENAME_KEY := TRUE;
          
END_FUNCTION

{attribute 'reflection'}
FUNCTION_BLOCK FB_HVAC_BURNER_MQTT EXTENDS FB_MQTT_BASE
  VAR_OUTPUT
    OUT : BOOL;
  END_VAR
  VAR
    {attribute 'noinit'}
    {attribute 'instance-path'}
    sInstancePath : STRING(GVL_MQTT.MQTT_TOPIC_LEN);  (* Refelection: object's full instance name *)
    bStartup : BOOL := TRUE;
    fbActuator : OSCAT_BUILDING.ACTUATOR_PUMP;
    MIN_ONTIME : TIME;
    MIN_OFFTIME : TIME;
    RUNTIME : UDINT;
    CYCLES : UDINT;
  END_VAR
  VAR PERSISTENT
    bPreviousState : BOOL;  (* To retain output state through powercycles *)
  END_VAR
  VAR_INPUT
    IN : BOOL;
  END_VAR

            (* --- self-wiring prologue ----------------------------------------------------
   Makes the InitMqtt and InitMqttDiscovery* calls optional. Set FriendlyName at
   the declaration site and this block wires itself from GVL_MQTT on its
   first cyclic call, then announces itself to Home Assistant.

   Deliberately in the body rather than in FB_init: it dereferences GVL members
   and reads the reflection instance path, and doing that during initialisation
   would rely on an ordering nothing enforces and the compiler cannot check. The
   body is the same lifecycle phase the init actions used, so this is not merely
   safe, it is the phase that already works today.

   The wiring calls this block's own unmodified InitMqtt / InitMqttDiscovery*
   methods, so anything published - topics and discovery JSON alike - is produced
   by exactly the code that produces it today. Only the trigger moved.

   Dormant while FriendlyName is empty, so existing projects and existing call
   sites keep working untouched.

   A block wired this way MUST be called cyclically. An instance whose body never
   runs is now unwired and absent from Home Assistant, where the init action used
   to wire it regardless. Nothing warns about that.  *)
IF FriendlyName <> '' THEN

	IF NOT bInitMqttDone THEN
		THIS^.InitMqtt(
			MQTTPublishPrefix := ADR(GVL_MQTT.MqttPubHVACPrefix),
			pMqttPublishQueue := ADR(GVL_MQTT.fbMqttPublishQueue));
	END_IF

	IF bInitMqttDone AND NOT bInitMqttDiscoveryDone THEN
		THIS^.InitMqttDiscovery(
			Device := ADR(GVL_MQTT.PLC_Device),
			Name := FriendlyName);
	END_IF

END_IF

fbActuator(
	IN := IN,
	MANUAL := FALSE,
	RST := FALSE,
	MIN_ONTIME := MIN_ONTIME,
	MIN_OFFTIME := MIN_OFFTIME,
	RUN_EVERY := T#0S,
	PUMP => OUT,
	RUNTIME := RUNTIME,
	CYCLES := CYCLES);
	
	
IF ((bPreviousState <> OUT) OR bStartup) AND bInitMqttDone THEN
	pMqttPublishQueue^.AddMessageOn(Lane := GVL_MQTT.MQTT_LANE_HVAC,
		Payload := BOOL_TO_STRING(OUT),
		Topic := sMQTTPublishTopic,
		Qos := MQTT.QoS.ExactlyOnce,
		MqttRetain := TRUE
	);	
	bStartup:=FALSE;
END_IF	

bPreviousState := OUT;
          

METHOD InitMqtt
  VAR_INPUT
    MQTTPublishPrefix : POINTER TO STRING;
    pMqttPublishQueue : POINTER TO FB_MQTT_PUBLISH_QUEUE;
  END_VAR
                  SUPER^._sInstancePath := THIS^.sInstancePath; // Due to reflection its location is important

(*pass trough*)
THIS^.pMqttPublishQueue := pMqttPublishQueue;
THIS^.psMqttPublishTopicPrefix:=MQTTPublishPrefix;
SUPER^.InitBaseMqtt();

                
END_METHOD

METHOD InitMqttDiscovery
  VAR_INPUT
    Device : POINTER TO FB_PLC_MQTT_DISCOVERY_DEVICE;
    Name : STRING(255);
    DeviceClass : STRING(100) := 'heat';
    overruleId : STRING(255) := '';
  END_VAR
  VAR
    id : STRING(255);
  END_VAR
                  IF bInitMqttDone AND NOT bInitMqttDiscoveryDone THEN
	
	id := SUPER^.ResolveEntityId(overruleId);
	
	Device^.CreateBinarySensorEntity(
		Id := id,
		Name := name,
		StateTopic := THIS^.sMQTTPublishTopic,
		PayloadOn := 'TRUE',
		PayloadOff := 'FALSE',
		DeviceClass := DeviceClass);
		
	bInitMqttDiscoveryDone := TRUE;
END_IF		
                
END_METHOD

(* FB_Init is always available implicitly and it is used primarily for initialization. The return value is not evaluated. For a specific influence, you can also declare the methods explicitly and provide additional code there with the standard initialization code. You can evaluate the return value. *)
METHOD FB_init : BOOL
  VAR_INPUT
    bInitRetains : BOOL;  (* TRUE: the retain variables are initialized (reset warm / reset cold) *)
    bInCopyCode : BOOL;  (* TRUE: the instance will be copied to the copy code afterward (online change) *)
    MIN_ONTIME : TIME;
    MIN_OFFTIME : TIME;
  END_VAR
                  THIS^.MIN_ONTIME := MIN_ONTIME;
THIS^.MIN_OFFTIME := MIN_OFFTIME;
                
END_METHOD
END_FUNCTION_BLOCK

{attribute 'reflection'}
FUNCTION_BLOCK FB_HVAC_COLLECTOR_MQTT EXTENDS FB_MQTT_BASE
  VAR CONSTANT
    ciValveCount : INT := 8;  (* Circuits on the manifold. A hardware fact rather than a tuning knob, and the one place the count is written for this block. A caller that passes a valve name array has to spell the same bound - see CollectorValveNames in PRG_HVAC. *)
    casValveNames : ARRAY[1..ciValveCount] OF STRING(8) := ['VALVE_1', 'VALVE_2', 'VALVE_3', 'VALVE_4', 'VALVE_5', 'VALVE_6', 'VALVE_7', 'VALVE_8'];  (* Spelled out instead of built with INT_TO_STRING at runtime. These strings are the published topic suffix AND the tail of the Home Assistant entity id, so a formatting surprise - a padded ' 1', a different width - would silently rename every valve entity in Home Assistant and orphan the old ones. *)
  END_VAR
  VAR_INPUT
    THERMOSTAT : ARRAY[1..ciValveCount] OF BOOL;  (* Heat demand, one element per circuit. The index IS the valve number as it appears on MQTT and in the entity id: THERMOSTAT[1] drives VALVE[1], which publishes to <topic>/Valves/VALVE_1. Renumbering these renames Home Assistant entities, so the indices are part of the interface, not an implementation detail. *)
    PUMP_MIN_ONTIME_ACTIVE : BOOL;  (* TRUE while the pump this manifold feeds is still running out its minimum on-time after the demand that started it has gone. Wire it to the pump's MIN_ONTIME_ACTIVE output: while it is set, the circuits that were last flowing are held open so the pump always has somewhere to push water. Optional, and FALSE is the old behaviour exactly - an existing call site that does not wire it keeps compiling and keeps closing its valves the moment demand ends. It is only safe to leave unwired if the pump's minimum on-time is shorter than the time the valves take to close. *)
  END_VAR
  VAR_OUTPUT
    VALVE : ARRAY[1..ciValveCount] OF BOOL;
    PUMP : BOOL;
  END_VAR
  VAR
    {attribute 'noinit'}
    {attribute 'instance-path'}
    sInstancePath : STRING(GVL_MQTT.MQTT_TOPIC_LEN);  (* Refelection: object's full instance name *)
    bStartup : BOOL := TRUE;
    fbPumpDelay : TON;
    bHeatRequest : BOOL;
    ValveCycleTime : TIME;
    abValveHeld : ARRAY[1..ciValveCount] OF BOOL;  (* Which circuits were flowing when the manifold last had demand. The hold re-opens exactly these, so the water keeps going where it was already going instead of through whichever circuit happens to be index 1. *)
    afbRTrigValve : ARRAY[1..ciValveCount] OF R_TRIG;
    afbFTrigValve : ARRAY[1..ciValveCount] OF F_TRIG;
    iI : INT;
  END_VAR

            // What the circuits are asking for. Built from THERMOSTAT and deliberately NOT from
// VALVE - see the interlock note below, where that distinction is the whole point.
bHeatRequest := FALSE;
FOR iI := 1 TO ciValveCount DO
	bHeatRequest := bHeatRequest OR THERMOSTAT[iI];
END_FOR

// Valves are NC: a valve is powered - open - exactly when its own circuit asks for
// heat, and closed otherwise.
//
// The exception is the interlock: FB_HVAC_PUMP_MQTT holds its output for MIN_ONTIME
// after its IN drops, so a manifold that closes the instant demand ends leaves the
// pump turning against shut valves. Whether that became a real dead-head depended on
// two timings configured on two different blocks - ValveCycleTime here against the
// pump's MIN_ONTIME there - with nothing in the code relating them. So while
// PUMP_MIN_ONTIME_ACTIVE is set, the circuits that were last flowing stay open and
// the pump keeps a path. This is requirement 2.3 in PRG_HVAC.HVAC_RUN, written down
// when this chain was designed and not implemented until now.
//
// The hold cannot latch on. It re-opens valves, but bHeatRequest stays FALSE, so
// this block never re-requests the pump: the pump's minimum on-time expires,
// PUMP_MIN_ONTIME_ACTIVE clears and the valves close. Building bHeatRequest from
// VALVE[] instead would close that loop and hold the pump on for ever. That used to
// be an identity - every VALVE[iI] was THERMOSTAT[iI], so the two ORs were the same
// value, and a comment here said so - and it is not an identity any more. Do not
// simplify it back.
IF bHeatRequest THEN
	FOR iI := 1 TO ciValveCount DO
		VALVE[iI] := THERMOSTAT[iI];
		abValveHeld[iI] := THERMOSTAT[iI];
	END_FOR
ELSE
	// No circuit is asking for heat: the valves are shut unless the pump is still
	// running out its minimum on-time, in which case the ones that were flowing
	// stay open until it stops.
	FOR iI := 1 TO ciValveCount DO
		VALVE[iI] := PUMP_MIN_ONTIME_ACTIVE AND abValveHeld[iI];
	END_FOR
END_IF

// Pump should only start when valves had time to switch to their correct position
fbPumpDelay(IN := bHeatRequest,
	PT := ValveCycleTime);

PUMP := bHeatRequest AND fbPumpDelay.Q;

// Detect edges on valves for MQTT messaging, and publish only the ones that moved.
// The topics are retained because Home Assistant reads them on reconnect, which is
// also why bStartup forces a publish of all eight on the first cycle after init.
// A valve held open by the interlock publishes TRUE for as long as it is held, which
// is what Home Assistant should see: the valve really is open.
FOR iI := 1 TO ciValveCount DO
	afbRTrigValve[iI](CLK := VALVE[iI]);
	afbFTrigValve[iI](CLK := VALVE[iI]);

	IF ((afbRTrigValve[iI].Q OR afbFTrigValve[iI].Q) OR bStartup) AND bInitMqttDone THEN
		pMqttPublishQueue^.AddMessageOn(Lane := GVL_MQTT.MQTT_LANE_HVAC,
			Payload := BOOL_TO_STRING(VALVE[iI]),
			Topic := CONCAT(sMQTTPublishTopic, CONCAT('/Valves/', casValveNames[iI])),
			Qos := MQTT.QoS.ExactlyOnce,
			MqttRetain := TRUE
		);
	END_IF
END_FOR

bStartup := FALSE;

          

METHOD InitMqtt
  VAR_INPUT
    MQTTPublishPrefix : POINTER TO STRING;
    pMqttPublishQueue : POINTER TO FB_MQTT_PUBLISH_QUEUE;
  END_VAR
                  SUPER^._sInstancePath := THIS^.sInstancePath; // Due to reflection its location is important

(*pass trough*)
THIS^.pMqttPublishQueue := pMqttPublishQueue;
THIS^.psMqttPublishTopicPrefix:=MQTTPublishPrefix;
SUPER^.InitBaseMqtt();

                
END_METHOD

METHOD InitMqttDiscovery
  VAR_INPUT
    Device : POINTER TO FB_PLC_MQTT_DISCOVERY_DEVICE;
    NameValve : ARRAY[1..ciValveCount] OF STRING(100);  (* One name per circuit, indexed as THERMOSTAT and VALVE are. An empty name means that circuit is not wired to anything and no Home Assistant entity is announced for it - which is how six of the eight stay invisible on the one instance this project has. *)
    DeviceClass : STRING(100) := 'water';
  END_VAR
  VAR
    id : STRING(255);
    iI : INT;
  END_VAR
                  IF bInitMqttDone AND NOT bInitMqttDiscoveryDone THEN

	FOR iI := 1 TO ciValveCount DO
		IF NOT(CommonTypesAndFunctions.StrEquals(str1:= ADR(NameValve[iI]), str2:= ADR(''))) THEN
			id := CONCAT(CONCAT(CONCAT(THIS^.DeviceName,'_'), THIS^.psInstanceNamePt^), CONCAT('_', THIS^.casValveNames[iI]));

			Device^.CreateValveStateEntity(
				Id := id,
				Name := NameValve[iI],
				StateTopic := CONCAT(THIS^.sMQTTPublishTopic, CONCAT('/Valves/', THIS^.casValveNames[iI])),
				StateOpen := 'TRUE',
				StateClosed := 'FALSE',
				DeviceClass := DeviceClass);
		END_IF
	END_FOR

	bInitMqttDiscoveryDone := TRUE;
END_IF

                
END_METHOD

(* FB_Init is always available implicitly and it is used primarily for initialization. The return value is not evaluated. For a specific influence, you can also declare the methods explicitly and provide additional code there with the standard initialization code. You can evaluate the return value. *)
METHOD FB_init : BOOL
  VAR_INPUT
    bInitRetains : BOOL;  (* TRUE: the retain variables are initialized (reset warm / reset cold) *)
    bInCopyCode : BOOL;  (* TRUE: the instance will be copied to the copy code afterward (online change) *)
    ValveCycleTime : TIME;
  END_VAR
                  THIS^.ValveCycleTime := ValveCycleTime;
                
END_METHOD
END_FUNCTION_BLOCK

{attribute 'reflection'}
FUNCTION_BLOCK FB_HVAC_PUMP_MQTT EXTENDS FB_MQTT_BASE
  VAR_OUTPUT
    PUMP : BOOL;
    HEAT_REQUEST : BOOL;  (* Alias of PUMP, kept deliberately: PRG_HVAC ORs both pumps' HEAT_REQUEST into the gas burner's demand input, so this is the name that expresses "this pump is asking for heat" at the call site. *)
    MIN_ONTIME_ACTIVE : BOOL;
  END_VAR
  VAR
    {attribute 'noinit'}
    {attribute 'instance-path'}
    sInstancePath : STRING(GVL_MQTT.MQTT_TOPIC_LEN);  (* Refelection: object's full instance name *)
    bStartup : BOOL := TRUE;
    fbActuator : OSCAT_BUILDING.ACTUATOR_PUMP;
    MIN_ONTIME : TIME;
    fbMinOntimeTimer : TON;
    MIN_OFFTIME : TIME;
    RUNTIME : UDINT;  (* Maintained by the OSCAT actuator and currently consumed by nobody. Left in place rather than deleted: these are pump lifetime statistics, and the useful fix is to publish them as diagnostic sensors, not to drop them. Note they are not persistent, so they count from the last download rather than for the life of the pump. *)
    CYCLES : UDINT;
  END_VAR
  VAR PERSISTENT
    bPreviousState : BOOL;  (* To retain output state through powercycles *)
  END_VAR
  VAR_INPUT
    IN : BOOL;
  END_VAR

            (* --- self-wiring prologue ----------------------------------------------------
   Makes the InitMqtt and InitMqttDiscovery* calls optional. Set FriendlyName at
   the declaration site and this block wires itself from GVL_MQTT on its
   first cyclic call, then announces itself to Home Assistant.

   Deliberately in the body rather than in FB_init: it dereferences GVL members
   and reads the reflection instance path, and doing that during initialisation
   would rely on an ordering nothing enforces and the compiler cannot check. The
   body is the same lifecycle phase the init actions used, so this is not merely
   safe, it is the phase that already works today.

   The wiring calls this block's own unmodified InitMqtt / InitMqttDiscovery*
   methods, so anything published - topics and discovery JSON alike - is produced
   by exactly the code that produces it today. Only the trigger moved.

   Dormant while FriendlyName is empty, so existing projects and existing call
   sites keep working untouched.

   A block wired this way MUST be called cyclically. An instance whose body never
   runs is now unwired and absent from Home Assistant, where the init action used
   to wire it regardless. Nothing warns about that.  *)
IF FriendlyName <> '' THEN

	IF NOT bInitMqttDone THEN
		THIS^.InitMqtt(
			MQTTPublishPrefix := ADR(GVL_MQTT.MqttPubHVACPrefix),
			pMqttPublishQueue := ADR(GVL_MQTT.fbMqttPublishQueue));
	END_IF

	IF bInitMqttDone AND NOT bInitMqttDiscoveryDone THEN
		THIS^.InitMqttDiscovery(
			Device := ADR(GVL_MQTT.PLC_Device),
			Name := FriendlyName);
	END_IF

END_IF

fbMinOntimeTimer(IN := IN, PT := MIN_ONTIME);
MIN_ONTIME_ACTIVE := NOT(fbMinOntimeTimer.Q) AND PUMP;

fbActuator(
	IN := IN,
	MANUAL := FALSE,
	RST := FALSE,
	MIN_ONTIME := MIN_ONTIME,
	MIN_OFFTIME := MIN_OFFTIME,
	RUN_EVERY := T#0S,
	PUMP => PUMP,
	RUNTIME := RUNTIME,
	CYCLES := CYCLES);
	
//Timer to keep track of ontime

HEAT_REQUEST := PUMP;	
	
IF ((bPreviousState <> PUMP) OR bStartup) AND bInitMqttDone THEN
	pMqttPublishQueue^.AddMessageOn(Lane := GVL_MQTT.MQTT_LANE_HVAC,
		Payload := BOOL_TO_STRING(PUMP),
		Topic := sMQTTPublishTopic,
		Qos := MQTT.QoS.ExactlyOnce,
		MqttRetain := TRUE
	);	
	bStartup:=FALSE;
END_IF	

bPreviousState := PUMP;
          

METHOD InitMqtt
  VAR_INPUT
    MQTTPublishPrefix : POINTER TO STRING;
    pMqttPublishQueue : POINTER TO FB_MQTT_PUBLISH_QUEUE;
  END_VAR
                  SUPER^._sInstancePath := THIS^.sInstancePath; // Due to reflection its location is important

(*pass trough*)
THIS^.pMqttPublishQueue := pMqttPublishQueue;
THIS^.psMqttPublishTopicPrefix:=MQTTPublishPrefix;
SUPER^.InitBaseMqtt();

                
END_METHOD

METHOD InitMqttDiscovery
  VAR_INPUT
    Device : POINTER TO FB_PLC_MQTT_DISCOVERY_DEVICE;
    Name : STRING(255);
    DeviceClass : STRING(100) := 'heat';
    overruleId : STRING(255) := '';
  END_VAR
  VAR
    id : STRING(255);
  END_VAR
                  IF bInitMqttDone AND NOT bInitMqttDiscoveryDone THEN
	
	id := SUPER^.ResolveEntityId(overruleId);
	
	Device^.CreateBinarySensorEntity(
		Id := id,
		Name := name,
		StateTopic := THIS^.sMQTTPublishTopic,
		PayloadOn := 'TRUE',
		PayloadOff := 'FALSE',
		DeviceClass := DeviceClass);
		
	bInitMqttDiscoveryDone := TRUE;
END_IF		
                
END_METHOD

(* FB_Init is always available implicitly and it is used primarily for initialization. The return value is not evaluated. For a specific influence, you can also declare the methods explicitly and provide additional code there with the standard initialization code. You can evaluate the return value. *)
METHOD FB_init : BOOL
  VAR_INPUT
    bInitRetains : BOOL;  (* TRUE: the retain variables are initialized (reset warm / reset cold) *)
    bInCopyCode : BOOL;  (* TRUE: the instance will be copied to the copy code afterward (online change) *)
    MIN_ONTIME : TIME;
    MIN_OFFTIME : TIME;
  END_VAR
                  THIS^.MIN_ONTIME := MIN_ONTIME;
THIS^.MIN_OFFTIME := MIN_OFFTIME;
                
END_METHOD
END_FUNCTION_BLOCK

{attribute 'reflection'}
FUNCTION_BLOCK FB_HVAC_THERMOSTAT_MQTT EXTENDS FB_MQTT_BASE IMPLEMENTS MQTT.MQTT_SUBSCRIBE_CALLBACK
  VAR_OUTPUT
    OUT : BOOL;
  END_VAR
  VAR
    {attribute 'noinit'}
    {attribute 'instance-path'}
    sInstancePath : STRING(GVL_MQTT.MQTT_TOPIC_LEN);  (* Refelection: object's full instance name *)
    bStartup : BOOL := TRUE;
    MinAllowedTemp : REAL := 12;
    MaxAllowedTemp : REAL := 30;
    Hysteresis : REAL := 0.5;  (* Zero would make this a bare comparison against the setpoint, and on a 50 ms task the output chatters at the setpoint - each flip a retained QoS 2 publish. 0.5 matches the TempStep the climate entity is announced with, so the deadband is the smallest step Home Assistant can ask for. *)
    rPreviousTemp : REAL;
    rPreviousHum : REAL;
    bSensorFault : BOOL;  (* Latches this scan's verdict on the temperature reading. *)
    bPreviousFault : BOOL;
  END_VAR
  VAR PERSISTENT
    rDesiredTemp : REAL;  (* To retain output state through powercycles *)
    bPreviousState : BOOL;
    eHvacMode : E_HVAC_MODE;
  END_VAR
  VAR_INPUT
    MEASURED_TEMP : REAL;
    MEASURED_HUM : REAL;
    ENABLED : BOOL := TRUE;
    SENSOR_VALID : BOOL := TRUE;  (* Wire this from the temperature source's own health outputs, e.g. SENSOR_VALID := sensor.DataAvailable AND NOT sensor.Error Defaults TRUE so existing call sites behave as before, but leaving it out means the thermostat is trusting a reading it cannot vouch for. *)
  END_VAR

            (* --- self-wiring prologue ----------------------------------------------------
   Makes the InitMqtt and InitMqttDiscovery* calls optional. Set FriendlyName at
   the declaration site and this block wires itself from GVL_MQTT on its
   first cyclic call, then announces itself to Home Assistant.

   Deliberately in the body rather than in FB_init: it dereferences GVL members
   and reads the reflection instance path, and doing that during initialisation
   would rely on an ordering nothing enforces and the compiler cannot check. The
   body is the same lifecycle phase the init actions used, so this is not merely
   safe, it is the phase that already works today.

   The wiring calls this block's own unmodified InitMqtt / InitMqttDiscovery*
   methods, so anything published - topics and discovery JSON alike - is produced
   by exactly the code that produces it today. Only the trigger moved.

   Dormant while FriendlyName is empty, so existing projects and existing call
   sites keep working untouched.

   A block wired this way MUST be called cyclically. An instance whose body never
   runs is now unwired and absent from Home Assistant, where the init action used
   to wire it regardless. Nothing warns about that.  *)
IF FriendlyName <> '' THEN

	IF NOT bInitMqttDone THEN
		THIS^.InitMqtt(
			MQTTPublishPrefix := ADR(GVL_MQTT.MqttPubHVACPrefix),
			MQTTSubscribePrefix := ADR(GVL_MQTT.MqttSubHVACPrefix),
			pMqttPublishQueue := ADR(GVL_MQTT.fbMqttPublishQueue),
			pMqttCallbackCollector := ADR(GVL_MQTT.collector_FB_HVAC_MQTT));
	END_IF

	IF bInitMqttDone AND NOT bInitMqttDiscoveryDone THEN
		THIS^.InitMqttDiscovery(
			Device := ADR(GVL_MQTT.PLC_Device),
			Name := FriendlyName,
			TempStep := 0.5);
	END_IF

END_IF

(* Refuse to act on a reading we cannot trust. Note the plausibility window
   alone would NOT catch this project's actual failure: 0.0 is a perfectly
   plausible temperature, so a dead sensor is only detectable via SENSOR_VALID.
   The window catches garbage from a mis-scaled or corrupted transfer. *)
bSensorFault := NOT SENSOR_VALID OR MEASURED_TEMP <= -50 OR MEASURED_TEMP >= 80;

IF bSensorFault THEN
	(* Fail safe: no heat demand on a suspect sensor. For a heating system this is
	   the branch that matters - the alternative is calling for heat forever. *)
	OUT := FALSE;
ELSIF NOT ENABLED OR eHvacMode = E_HVAC_MODE.off THEN
	OUT := FALSE;
ELSIF MEASURED_TEMP > MaxAllowedTemp THEN
	OUT := FALSE;
ELSIF ENABLED AND eHvacMode = E_HVAC_MODE.auto AND MEASURED_TEMP < MinAllowedTemp THEN
	OUT := TRUE;
ELSIF ENABLED AND eHvacMode = E_HVAC_MODE.auto AND OUT AND MEASURED_TEMP > (MinAllowedTemp + Hysteresis) THEN
	OUT := FALSE;
ELSIF ENABLED AND eHvacMode = E_HVAC_MODE.heat AND MEASURED_TEMP < (rDesiredTemp - Hysteresis) THEN
	OUT := TRUE;
ELSIF ENABLED AND eHvacMode = E_HVAC_MODE.heat AND MEASURED_TEMP > (rDesiredTemp + Hysteresis) THEN
	OUT := FALSE;
END_IF

IF bStartup AND bInitMqttDone THEN
	pMqttPublishQueue^.AddMessageOn(Lane := GVL_MQTT.MQTT_LANE_HVAC,
		Payload := REAL_TO_STRING(MaxAllowedTemp),
		Topic := CONCAT(sMQTTPublishTopic, '/MAX_TEMP'),
		Qos := MQTT.QoS.ExactlyOnce,
		MqttRetain := TRUE
	);	
	pMqttPublishQueue^.AddMessageOn(Lane := GVL_MQTT.MQTT_LANE_HVAC,
		Payload := REAL_TO_STRING(MinAllowedTemp),
		Topic := CONCAT(sMQTTPublishTopic, '/MIN_TEMP'),
		Qos := MQTT.QoS.ExactlyOnce,
		MqttRetain := TRUE
	);
	pMqttPublishQueue^.AddMessageOn(Lane := GVL_MQTT.MQTT_LANE_HVAC,
		Payload := TO_STRING(eHvacMode),
		Topic := CONCAT(sMQTTPublishTopic, '/MODE'),
		Qos := MQTT.QoS.ExactlyOnce,
		MqttRetain := TRUE
	);	
	pMqttPublishQueue^.AddMessageOn(Lane := GVL_MQTT.MQTT_LANE_HVAC,
		Payload := REAL_TO_STRING(rDesiredTemp),
		Topic := CONCAT(sMQTTPublishTopic, '/DESIRED_TEMP'),
		Qos := MQTT.QoS.ExactlyOnce,
		MqttRetain := TRUE
	);	
END_IF

IF ((bPreviousState <> OUT) OR bStartup) AND bInitMqttDone THEN
	pMqttPublishQueue^.AddMessageOn(Lane := GVL_MQTT.MQTT_LANE_HVAC,
		Payload := BOOL_TO_STRING(OUT),
		Topic := sMQTTPublishTopic,
		Qos := MQTT.QoS.ExactlyOnce,
		MqttRetain := TRUE
	);	
END_IF	
IF ((rPreviousTemp <> MEASURED_TEMP) OR bStartup) AND bInitMqttDone THEN
	pMqttPublishQueue^.AddMessageOn(Lane := GVL_MQTT.MQTT_LANE_HVAC,
		Payload := REAL_TO_STRING(MEASURED_TEMP),
		Topic := CONCAT(sMQTTPublishTopic, '/TEMP'),
		Qos := MQTT.QoS.ExactlyOnce,
		MqttRetain := TRUE
	);
END_IF

IF ((rPreviousHum <> MEASURED_HUM) OR bStartup) AND bInitMqttDone THEN
	pMqttPublishQueue^.AddMessageOn(Lane := GVL_MQTT.MQTT_LANE_HVAC,
		Payload := REAL_TO_STRING(MEASURED_HUM),
		Topic := CONCAT(sMQTTPublishTopic, '/HUM'),
		Qos := MQTT.QoS.ExactlyOnce,
		MqttRetain := TRUE
	);	
END_IF	


IF ((bPreviousFault <> bSensorFault) OR bStartup) AND bInitMqttDone THEN
	pMqttPublishQueue^.AddMessageOn(Lane := GVL_MQTT.MQTT_LANE_HVAC,
		Payload := BOOL_TO_STRING(bSensorFault),
		Topic := CONCAT(sMQTTPublishTopic, '/FAULT'),
		Qos := MQTT.QoS.ExactlyOnce,
		MqttRetain := TRUE
	);
END_IF
bPreviousFault := bSensorFault;

bStartup:=FALSE;
rPreviousTemp := MEASURED_TEMP;
rPreviousHum := MEASURED_HUM;
bPreviousState := OUT;
          

METHOD InitMqtt
  VAR_INPUT
    MQTTPublishPrefix : POINTER TO STRING;
    MQTTSubscribePrefix : POINTER TO STRING;
    pMqttPublishQueue : POINTER TO FB_MQTT_PUBLISH_QUEUE;
    pMqttCallbackCollector : POINTER TO MQTT.CallbackCollector;
  END_VAR
                  SUPER^._sInstancePath := THIS^.sInstancePath; // Due to reflection its location is important

(*pass trough*)
THIS^.pMqttPublishQueue := pMqttPublishQueue;
THIS^.psMqttPublishTopicPrefix:=MQTTPublishPrefix;
THIS^.psMqttSubscribeTopicPrefix:=MQTTSubscribePrefix;
THIS^.pMqttPublishQueue:=pMqttPublishQueue;

SUPER^.InitBaseMqtt();
pMqttCallbackCollector^.put(instance:= THIS^); // register the FB agains the collector so mqtt events can be received


                
END_METHOD

METHOD InitMqttDiscovery
  VAR_INPUT
    Device : POINTER TO FB_PLC_MQTT_DISCOVERY_DEVICE;
    Name : STRING(255);
    TempStep : REAL;
    overruleId : STRING(255) := '';
  END_VAR
  VAR
    id : STRING(255);
  END_VAR
                  IF bInitMqttDone AND NOT bInitMqttDiscoveryDone THEN
	
	id := SUPER^.ResolveEntityId(overruleId);
	
	Device^.CreateClimateEntity(		
		Id := id,
		Name := name,
		InitialDesiredTemperature := REAL_TO_INT(rDesiredTemp),
		CurrentTemperatureTopic :=  CONCAT(sMQTTPublishTopic, '/TEMP'),
		CurrentHumidityTopic := CONCAT(sMQTTPublishTopic, '/HUM'),
		ModeCommandTopic := CONCAT(THIS^.sMQTTSubscribeTopic, '/MODE'),
		ModeStateTopic := CONCAT(THIS^.sMQTTPublishTopic, '/MODE'),
		TemperatureCommandTopic := CONCAT(THIS^.sMQTTSubscribeTopic, '/DESIRED_TEMP') ,
		TemperatureStateTopic := CONCAT(THIS^.sMQTTPublishTopic, '/DESIRED_TEMP'),
		TempStep := TempStep);
		
	bInitMqttDiscoveryDone := TRUE;
END_IF		
                
END_METHOD

METHOD PublishReceived : BOOL
  VAR_INPUT
    Data : MQTT.CALLBACK_DATA;  (* Collection of recived Data *)
  END_VAR
                  //first check if Mqtt is initialized, otherwise do nothing
IF NOT(bInitMqttDone) THEN
	//mark the interface call from the collector as done
	PublishReceived := TRUE;
//check if the packet is for this FB
ELSIF CONCAT(sMQTTSubscribeTopic,'/DESIRED_TEMP') =  Data.TopicOut^ THEN
	//mark the interface call from the collector as done
	PublishReceived := TRUE;
	//check if temp is numeric, then assign it;
	IF OSCAT_BASIC.IS_CC(str:= Data.PayloadString^,cmp:='0123456789.') THEN
		 // temperature requested higher then max allowed temp; set to max allowed temp
		 IF STRING_TO_REAL(Data.PayloadString^) > THIS^.MaxAllowedTemp THEN
			 THIS^.rDesiredTemp := THIS^.MaxAllowedTemp;		 
			 THIS^.pMqttPublishQueue^.AddMessageOn(Lane := GVL_MQTT.MQTT_LANE_HVAC,
				Payload := REAL_TO_STRING(THIS^.MaxAllowedTemp),
				Topic := CONCAT(sMQTTPublishTopic, '/DESIRED_TEMP'),
				Qos := MQTT.QoS.ExactlyOnce,
				MqttRetain := TRUE
			);
		 // temperature requested lower then min allowed temp: set to min allowed temp
		 ELSIF STRING_TO_REAL(Data.PayloadString^) < THIS^.MinAllowedTemp THEN
			 THIS^.rDesiredTemp := THIS^.MinAllowedTemp;			 
			 THIS^.pMqttPublishQueue^.AddMessageOn(Lane := GVL_MQTT.MQTT_LANE_HVAC,
				Payload := REAL_TO_STRING(THIS^.MinAllowedTemp),
				Topic := CONCAT(sMQTTPublishTopic, '/DESIRED_TEMP'),
				Qos := MQTT.QoS.ExactlyOnce,
				MqttRetain := TRUE
			);
		 ELSE
			 THIS^.rDesiredTemp := STRING_TO_REAL(Data.PayloadString^);			 
			 THIS^.pMqttPublishQueue^.AddMessageOn(Lane := GVL_MQTT.MQTT_LANE_HVAC,
				Payload := Data.PayloadString^,
				Topic := CONCAT(sMQTTPublishTopic, '/DESIRED_TEMP'),
				Qos := MQTT.QoS.ExactlyOnce,
				MqttRetain := TRUE
			);
		 END_IF
	END_IF
	
ELSIF CONCAT(sMQTTSubscribeTopic,'/MODE') =  Data.TopicOut^ THEN
	//mark the interface call from the collector as done
	PublishReceived := TRUE;
	//check if the mode is known and if so set it
	IF CommonTypesAndFunctions.StrEquals(str1:= Data.PayloadString, str2:= ADR('auto')) THEN
		THIS^.eHvacMode := E_HVAC_MODE.auto;		
	 	THIS^.pMqttPublishQueue^.AddMessageOn(Lane := GVL_MQTT.MQTT_LANE_HVAC,
			Payload := Data.PayloadString^,
			Topic := CONCAT(sMQTTPublishTopic, '/MODE'),
			Qos := MQTT.QoS.ExactlyOnce,
			MqttRetain := TRUE
		);
	ELSIF CommonTypesAndFunctions.StrEquals(str1:= Data.PayloadString, str2:= ADR('off')) THEN
		THIS^.eHvacMode := E_HVAC_MODE.off;		
	 	THIS^.pMqttPublishQueue^.AddMessageOn(Lane := GVL_MQTT.MQTT_LANE_HVAC,
			Payload := Data.PayloadString^,
			Topic := CONCAT(sMQTTPublishTopic, '/MODE'),
			Qos := MQTT.QoS.ExactlyOnce,
			MqttRetain := TRUE
		);
	ELSIF CommonTypesAndFunctions.StrEquals(str1:= Data.PayloadString, str2:= ADR('heat')) THEN
		THIS^.eHvacMode := E_HVAC_MODE.heat;		
	 	THIS^.pMqttPublishQueue^.AddMessageOn(Lane := GVL_MQTT.MQTT_LANE_HVAC,
			Payload := Data.PayloadString^,
			Topic := CONCAT(sMQTTPublishTopic, '/MODE'),
			Qos := MQTT.QoS.ExactlyOnce,
			MqttRetain := TRUE
		);
	END_IF;
END_IF 
                
END_METHOD

(* FB_Init is always available implicitly and it is used primarily for initialization. The return value is not evaluated. For a specific influence, you can also declare the methods explicitly and provide additional code there with the standard initialization code. You can evaluate the return value. *)
METHOD FB_init : BOOL
  VAR_INPUT
    bInitRetains : BOOL;  (* TRUE: the retain variables are initialized (reset warm / reset cold) *)
    bInCopyCode : BOOL;  (* TRUE: the instance will be copied to the copy code afterward (online change) *)
    MinAllowedTemp : REAL;
    MaxAllowedTemp : REAL;
    Hysteresis : REAL;
  END_VAR
                  THIS^.MinAllowedTemp := MinAllowedTemp;
THIS^.MaxAllowedTemp := MaxAllowedTemp;
THIS^.Hysteresis := Hysteresis;
                
END_METHOD
END_FUNCTION_BLOCK

FUNCTION_BLOCK FB_MQTT_BASE
  VAR
    _sInstancePath : STRING(GVL_MQTT.MQTT_TOPIC_LEN);
    psInstanceNamePt : POINTER TO STRING;
    DeviceName : STRING;
    bInitMqttDone : BOOL;
    psMqttPublishTopicPrefix : POINTER TO STRING;  (* Publish (Out); *)
    MqttPublishTopicSuffix : STRING(GVL_MQTT.MQTT_SUFFIX_LEN);
    sMQTTPublishTopic : STRING(GVL_MQTT.MQTT_TOPIC_LEN);
    psMqttSubscribeTopicPrefix : POINTER TO STRING;  (* Subscribe (In) *)
    sMqttSubscribeTopicSuffix : STRING(GVL_MQTT.MQTT_SUFFIX_LEN);
    sMQTTSubscribeTopic : STRING(GVL_MQTT.MQTT_TOPIC_LEN);
    pMqttPublishQueue : POINTER TO FB_MQTT_PUBLISH_QUEUE;
    bMqttHighRequest : BOOL;
    bMqttLowRequest : BOOL;
    MqttQos : MQTT.QoS := MQTT.QoS.ExactlyOnce;
    MqttRetain : BOOL := TRUE;
    fbComposeJSON : STRUCT_TO_JSON;  (* HA Discovery specific *)
    bInitMqttDiscoveryDone : BOOL := FALSE;
    bTopicTruncated : BOOL;  (* TRUE when a composed topic did not fit and was silently cut short. Read it to prove a deployment's naming scheme actually fits, which is otherwise invisible until Home Assistant shows an entity as unavailable. *)
  END_VAR
  VAR_INPUT
    FriendlyName : STRING(255) := '';  (* Human readable name shown in Home Assistant. Setting it is what switches a block to self-wiring: on its first cyclic call the block reaches into GVL_MQTT for its publish queue, topic prefixes and callback collector, and announces itself for discovery. Leave it empty and the block behaves exactly as before, wired only by an explicit InitMqtt / InitMqttDiscovery* call - which remain available for anything this declaration-only API cannot express, such as a second broker, a custom prefix, or a per-instance Home Assistant device. *)
    EntityType : E_MQTT_ENTITY := E_MQTT_ENTITY.Default;  (* Which Home Assistant platform to announce as. Default means "whatever this block has always announced as", so an existing project keeps its entity platform without naming it. A block announced as something other than its own default MUST say so here: FB_DO_BIN_001 is a binary output announced as a Light, and getting that wrong silently orphans the retained light/.../config topic and creates a new switch entity instead. *)
    RelayType : E_RELAY_TYPE := E_RELAY_TYPE.NO;  (* Which way round the contact this output drives sits: NO (the default) means the load is live when OUT is TRUE, NC means it is live when OUT is FALSE. It changes nothing in the PLC and everything in the discovery config, which swaps payload_on / payload_off so Home Assistant reports the state of the LOAD rather than of the coil. Get it wrong on an NC circuit and the entity reads exactly backwards, with nothing anywhere to flag it. NC is not exotic: it is how anything that must survive a dead controller is wired, sockets above all. Honoured only by blocks whose discovery methods take it - the binary and bistable outputs - and accepted and ignored elsewhere, the same way EntityType is on a block that can only be one thing. *)
  END_VAR

            
          

METHOD InitBaseMqtt
                  
(*Define instance names*)
psInstanceNamePt := CommonTypesAndFunctions.FindLastDot(ADR(_sInstancePath)) + 1;

DeviceName := LEFT(_sInstancePath,find(_sInstancePath, '.' )-1  ) ;

// Publish (Out);
IF	psMqttPublishTopicPrefix <> 0 THEN
	THIS^.MqttPublishTopicSuffix := psInstanceNamePt^;
	THIS^.sMQTTPublishTopic := CONCAT(psMqttPublishTopicPrefix^, THIS^.MqttPublishTopicSuffix);
END_IF

// Subscribe (In)
IF	psMqttSubscribeTopicPrefix <> 0 THEN
	THIS^.sMqttSubscribeTopicSuffix := psInstanceNamePt^;
	THIS^.sMQTTSubscribeTopic := CONCAT(psMqttSubscribeTopicPrefix^ ,THIS^.sMqttSubscribeTopicSuffix);
END_IF

(* Make truncation detectable. IEC cuts an over-long CONCAT short without any
   error, so without this the only symptom is an entity that never appears. *)
IF psMqttPublishTopicPrefix <> 0 THEN
	IF LEN(psMqttPublishTopicPrefix^) + LEN(THIS^.MqttPublishTopicSuffix) > GVL_MQTT.MQTT_TOPIC_LEN THEN
		THIS^.bTopicTruncated := TRUE;
	END_IF
END_IF
IF psMqttSubscribeTopicPrefix <> 0 THEN
	IF LEN(psMqttSubscribeTopicPrefix^) + LEN(THIS^.sMqttSubscribeTopicSuffix) > GVL_MQTT.MQTT_TOPIC_LEN THEN
		THIS^.bTopicTruncated := TRUE;
	END_IF
END_IF

(* The queue is dereferenced without a null check in every publishing block,
   so refuse to be initialised without one. The derived InitMqtt assigns
   THIS^.pMqttPublishQueue before calling this, which is why it can be read
   here. A block left uninitialised publishes nothing; one initialised with a
   null queue faults on its first publish instead. *)
IF THIS^.pMqttPublishQueue = 0 THEN
	RETURN;
END_IF

bInitMqttDone := TRUE;
                
END_METHOD

METHOD ResolveEntityId : STRING(255)
  VAR_INPUT
    overruleId : STRING(255) := '';  (* Pass an externally chosen id to override the derived one; empty means derive. *)
  END_VAR
                  (* The Home Assistant entity id. This rule used to be copy-pasted into every
   InitMqttDiscovery* method, so changing it - lower-casing it, stripping a
   prefix - meant 21 consistent edits, and one missed edit silently orphans
   entities in Home Assistant. *)
IF CommonTypesAndFunctions.StrEquals(str1:= ADR(overruleId), str2:= ADR('')) THEN
	ResolveEntityId := CONCAT(CONCAT(THIS^.DeviceName,'_'), THIS^.psInstanceNamePt^); // 'FB_DI_PB_003'
ELSE
	ResolveEntityId := overruleId; // 'MY_PH_GND_HALL_01'
END_IF
                
END_METHOD
END_FUNCTION_BLOCK

(* A ring buffer per producing task, drained by one consumer. Each lane is single-producer / single-consumer, which is the invariant the original design relied on and could not enforce: iPw of a lane is written only by the task that owns that lane, iPr only by the drain, and each side merely reads the other's index - a single aligned INT load on this 32-bit target, which cannot tear. No semaphore, so no priority inversion. What this fixes, and why it mattered: two tasks in AddMessage at once read the same iPw, wrote into the same slot and left a hybrid there - one message's topic carrying another's payload. On Bijbouw that showed up as a device publishing 'offline' it had never sent, three times per its own count against seventeen on the broker. Sharing one lane between tasks brings it straight back, so a producer that runs in its own task takes its own lane. Lanes hold the same total storage the single ring did. ST_MQTT_MESSAGE is about 1.8 kB, so the ring is already megabytes and a second instance was never an option on this hardware. *)
FUNCTION_BLOCK FB_MQTT_PUBLISH_QUEUE
  VAR_OUTPUT
    DroppedCount : UDINT;  (* Messages discarded because a lane was full. Without this, overflow is completely silent - and the DMX log flood made overflow easy to provoke. *)
  END_VAR
  VAR
    astFifo : ARRAY[0..ciLanes, 0..ciLaneN] OF ST_MQTT_MESSAGE;
    aiPr : ARRAY[0..ciLanes] OF INT;  (* Read index per lane. Advanced ONLY by GetMessage. *)
    aiPw : ARRAY[0..ciLanes] OF INT;  (* Write index per lane. Advanced ONLY by the task that owns the lane. *)
    iDrain : INT := 0;  (* Round-robin drain cursor, so a busy lane cannot starve a quiet one. *)
    iScan : INT;
  END_VAR
  VAR CONSTANT
    ciLanes : INT := 2;  (* Highest lane index. One per producing task: 0 MainTask, 1 the RS485 task, 2 HvacTask. GVL_MQTT.MQTT_LANE_* names them for the producers. *)
    ciLaneN : INT := 340;  (* Highest slot index within a lane. Chosen so that adding a lane does not add storage: 3 x 341 is the 1024 slots the single ring had. A slot is about 1.8 kB, so a lane costs roughly 600 kB and cannot just be added. *)
  END_VAR

            
          

METHOD GetMessage : ST_MQTT_MESSAGE
                  (* Round-robin across the lanes, so a loud producer cannot starve a quiet one.

   Copy the slot out before releasing it: advancing aiPr is what tells the
   producer the slot may be overwritten, so it has to be the last thing that
   happens. *)
FOR iScan := 0 TO ciLanes DO
	iDrain := iDrain + 1;
	IF iDrain > ciLanes THEN
		iDrain := 0;
	END_IF

	IF aiPr[iDrain] <> aiPw[iDrain] THEN
		GetMessage := astFifo[iDrain, aiPr[iDrain]];
		aiPr[iDrain] := OSCAT_BASIC.INC1(aiPr[iDrain], ciLaneN);
		RETURN;
	END_IF
END_FOR

                
END_METHOD

METHOD AddMessage
  VAR_INPUT
    Payload : STRING(1500);
    Topic : STRING(GVL_MQTT.MQTT_TOPIC_LEN);
    Qos : MQTT.QoS;
    MqttRetain : BOOL;
  END_VAR
                  (* The default lane. Anything that does not name one shares lane 0, which is
   correct only while those callers run in the same task - true today for
   MainTask, and the reason the RS485 blocks name lane 1 instead. *)
THIS^.AddMessageOn(Lane := 0,
				Payload := Payload,
				Topic := Topic,
				Qos := Qos,
				MqttRetain := MqttRetain);

                
END_METHOD

METHOD HasMessage : BOOL
                  (* Any lane with something in it. *)
HasMessage := FALSE;
FOR iScan := 0 TO ciLanes DO
	IF aiPr[iScan] <> aiPw[iScan] THEN
		HasMessage := TRUE;
		RETURN;
	END_IF
END_FOR

                
END_METHOD

METHOD IsFull : BOOL
                  (* Kept for callers that ask about the default lane. A lane reports full one
   slot early: that is what buys aiPr = aiPw its unambiguous 'empty' meaning. *)
IsFull := OSCAT_BASIC.INC1(aiPw[0], ciLaneN) = aiPr[0];

                
END_METHOD

(* Queue a message on a specific lane. A lane must be written by ONE task only. *)
METHOD AddMessageOn
  VAR_INPUT
    Lane : INT;  (* 0 for the default lane, 1 for the RS485 task. Out of range falls back to 0. *)
    Payload : STRING(1500);
    Topic : STRING(GVL_MQTT.MQTT_TOPIC_LEN);
    Qos : MQTT.QoS;
    MqttRetain : BOOL;
  END_VAR
  VAR
    iL : INT;
  END_VAR
                  (* Written straight into the slot. aiPw[iL] is advanced only once all four
   fields are in place, and GetMessage never reads a slot while aiPr = aiPw, so
   the drain cannot observe a half-written entry.

   Safe against a second writer ONLY because a lane has one. That is the whole
   point of the lane: two tasks sharing one would collide on aiPw exactly as
   they used to collide on the single iPw. *)
iL := Lane;
IF (iL < 0) OR (iL > ciLanes) THEN
	iL := 0;
END_IF

IF OSCAT_BASIC.INC1(aiPw[iL], ciLaneN) <> aiPr[iL] THEN
	astFifo[iL, aiPw[iL]].Payload := Payload;
	astFifo[iL, aiPw[iL]].Topic := Topic;
	astFifo[iL, aiPw[iL]].Qos := Qos;
	astFifo[iL, aiPw[iL]].MqttRetain := MqttRetain;
	(* Last: advancing the write index is what publishes the slot to the drain. *)
	aiPw[iL] := OSCAT_BASIC.INC1(aiPw[iL], ciLaneN);
ELSE
	DroppedCount := DroppedCount + 1;
END_IF

                
END_METHOD
END_FUNCTION_BLOCK

FUNCTION_BLOCK FB_MQTT_PUBLISH_WORKER
  VAR_OUTPUT
    SendDone : BOOL;
    SendErrorCount : UDINT;  (* Publishes abandoned on timeout. Each one used to retire this worker permanently; now it is released and this counts how often that happened. *)
  END_VAR
  VAR
    stLocalMqttMessage : ST_MQTT_MESSAGE;
    bInitDone : BOOL;
    bRequestToSend : BOOL;
    Send : BOOL;
    fbPublish : MQTT.MQTTPublish;
    fbSendTimeout : TON;  (* Bounds how long a single fbPublish may hold this worker. *)
    bSendOverdue : BOOL;  (* Latches an overdue publish so it is counted once rather than every cycle. Cleared when the worker accepts a new message. *)
  END_VAR

            //need to call fbPublish here because of FB nums
fbPublish(
	Topic:= ADR(stLocalMqttMessage.Topic), 
	PayloadString:= ADR(stLocalMqttMessage.Payload), 
	PublishAsString:= TRUE, 
	QoSIn:= stLocalMqttMessage.Qos, 
	MRetain:= stLocalMqttMessage.MqttRetain, 
	send:= Send);
	
IF NOT bInitDone THEN RETURN; END_IF

IF bRequestToSend THEN
	Send := TRUE;
	SendDone := FALSE;
END_IF

fbSendTimeout(IN := Send, PT := T#10S);

IF fbPublish.done THEN
	 SendDone := TRUE;
	 bRequestToSend:=FALSE;
	 Send:=FALSE;
	 fbSendTimeout(IN := FALSE);
ELSIF fbSendTimeout.Q AND NOT bSendOverdue THEN
	(* Count an overdue publish, but do NOT hand the worker back. Handing it back
	   is what poisoned the next message.

	   MqttPublish builds its packet once, on the rising edge of send: it captures
	   LEN(Topic) into MqttTopicLength and keeps only a POINTER to the topic, and
	   it clears dataBuild when the publish completes - not when the connection
	   drops, where it deliberately leaves the build standing so the packet is
	   re-sent on reconnect. A recycled worker therefore does not rebuild: the next
	   message reaches the library through that same pointer while the length stays
	   that of the previous topic, so a shorter topic publishes with a longer
	   length. The topic field runs past its terminator into NULs and the tail of
	   the topic before it, which is not a valid MQTT topic - a topic may not
	   contain U+0000 - and the broker answers by closing the connection.

	   Captured on the bench: a 30-character topic declared as 56 bytes, a broker
	   FIN 160 ms after CONNACK, and a reconnect loop nothing but restarting the
	   application could clear, because the poisoned build was replayed on every
	   new session.

	   SendDone now waits for fbPublish instead of for the clock. A worker holding
	   an unfinished publish through an outage finishes it on reconnect, when
	   MqttPublish re-sends the packet it already built, and rejoins the pool then. *)
	 SendErrorCount := SendErrorCount + 1;
	 bSendOverdue := TRUE;
END_IF
          

METHOD Init
  VAR_INPUT
    inputMQTT_IN_OUT : POINTER TO MQTT.MQTT_IN_OUT;  (* Pointer MQTTT exchange strucure *)
  END_VAR
                  fbPublish.SetMqttInOut(MQTT_IN_OUT := inputMQTT_IN_OUT^);

bInitDone := TRUE;
SendDone := TRUE;

                
END_METHOD

METHOD PublishMessage
  VAR_INPUT
    MqttMessage : ST_MQTT_MESSAGE;
  END_VAR
                  stLocalMqttMessage := MqttMessage;

bSendOverdue := FALSE;
bRequestToSend:=TRUE;
                
END_METHOD
END_FUNCTION_BLOCK

FUNCTION F_STRIP_JSON_ROOT : BOOL
  VAR_INPUT
    pJson : POINTER TO BYTE;  (* ADR(sJson) *)
    uiSize : UINT;  (* SIZEOF(sJson) *)
  END_VAR
  VAR
    diContentLen : DINT;
    diStart : DINT;
    diEnd : DINT;
    diI : DINT;
    bFoundStart : BOOL;
    bFoundEnd : BOOL;
  END_VAR

            
// Returns TRUE if successful, FALSE if the string could not be parsed.
// The result is written back into the string in-place.

F_STRIP_JSON_ROOT := FALSE;

// Find actual string length by scanning for null terminator
diContentLen := 0;
FOR diI := 0 TO UINT_TO_DINT(uiSize) - 1 DO
    IF pJson[diI] = 0 THEN
        diContentLen := diI;
        EXIT;
    END_IF
END_FOR

IF diContentLen < 5 THEN
    RETURN;
END_IF

// Find the first occurrence of ':{' (byte values 58 and 123)
bFoundStart := FALSE;
FOR diI := 0 TO diContentLen - 2 DO
    IF (pJson[diI] = 16#3A) AND (pJson[diI + 1] = 16#7B) THEN
        diStart := diI + 1; // index of the inner '{'
        bFoundStart := TRUE;
        EXIT;
    END_IF
END_FOR

IF NOT bFoundStart THEN
    RETURN;
END_IF

// Find the last '}' (byte value 125) scanning backwards
bFoundEnd := FALSE;
FOR diI := diContentLen - 1 TO 0 BY -1 DO
    IF pJson[diI] = 16#7D THEN
        diEnd := diI;
        bFoundEnd := TRUE;
        EXIT;
    END_IF
END_FOR

IF NOT bFoundEnd THEN
    RETURN;
END_IF

// diEnd must come after diStart. It does not on JSON that was truncated or was
// never well formed, and then diEnd - diStart is negative: DINT_TO_UDINT turns
// that into ~4 GB for SysMemMove, and pJson[diEnd - diStart] writes in front of
// the buffer. Neither reports anything.
IF diEnd <= diStart THEN
    RETURN;
END_IF

// diEnd is the outer '}', the inner object runs from diStart to diEnd - 1
// Move the inner content to the beginning of the buffer
SysMemMove(pDest := pJson, pSrc := ADR(pJson[diStart]), udiCount := DINT_TO_UDINT(diEnd - diStart));

// Null-terminate
pJson[diEnd - diStart] := 0;

F_STRIP_JSON_ROOT := TRUE;
          
END_FUNCTION

{attribute 'reflection'}
FUNCTION_BLOCK FB_1WIRE_MQTT_DISCOVERY_DEVICE EXTENDS FB_BASE_MQTT_DISCOVERY_DEVICE
  VAR
    manufacturer : STRING;
  END_VAR

            
          

METHOD init1WireDevice
  VAR_INPUT
    name : STRING;
    id : STRING;
    deviceAvailabilityTopic : STRING(GVL_MQTT.MQTT_TOPIC_LEN) := '';
    deviceDiagnosticTopic : STRING(GVL_MQTT.MQTT_TOPIC_LEN) := '';
  END_VAR
                  (* A 1-Wire sensor announces itself to Home Assistant as a device of its own, so
   its diagnostics belong to the sensor and not to the controller: both the Log
   entity and the diagnostic availability entity have to name the sensor's own
   topics. Both arguments are optional, so a call site that does not know its own
   topics keeps whatever FB_init supplied - which is the controller's. *)
IF bInit THEN
	bInit := FALSE;

	IF deviceAvailabilityTopic <> '' THEN
		THIS^.availabilityTopic2 := deviceAvailabilityTopic;
	END_IF

	IF deviceDiagnosticTopic <> '' THEN
		THIS^.MqttDiagnosticTopic := deviceDiagnosticTopic;
	END_IF

	SUPER^.initBaseDevice(
		Name := name,
		Identifiers := id,
		Manufacturer := Manufacturer,
		availabilityTopic := availabilityTopic1,
		availabilityTopic2 := THIS^.availabilityTopic2,
		availabilityOnline := availabilityOnline,
		availabilityOffline := availabilityOffline,
		MqttDiscoveryPrefix := MqttDiscoveryPrefix,
		MqttDiagnosticTopic := THIS^.MqttDiagnosticTopic,
		pMqttPublishQueue := pMqttPublishQueue);
END_IF

                
END_METHOD

(* FB_Init is always available implicitly and it is used primarily for initialization. The return value is not evaluated. For a specific influence, you can also declare the methods explicitly and provide additional code there with the standard initialization code. You can evaluate the return value. *)
METHOD FB_init : BOOL
  VAR_INPUT
    bInitRetains : BOOL;  (* TRUE: the retain variables are initialized (reset warm / reset cold) *)
    bInCopyCode : BOOL;  (* TRUE: the instance will be copied to the copy code afterward (online change) *)
    manufacturer : STRING;
    availabilityTopic : STRING(GVL_MQTT.MQTT_TOPIC_LEN);
    availabilityOnline : STRING;
    availabilityOffline : STRING;
    MqttDiscoveryPrefix : STRING;
    MqttDiagnosticTopic : STRING(GVL_MQTT.MQTT_TOPIC_LEN);
    pMqttPublishQueue : POINTER TO FB_MQTT_PUBLISH_QUEUE;
  END_VAR
                  THIS^.Manufacturer := Manufacturer;

THIS^.availabilityTopic1 := availabilityTopic;
THIS^.availabilityTopic2 := availabilityTopic;
THIS^.availabilityOnline := availabilityOnline;
THIS^.availabilityOffline := availabilityOffline;
THIS^.MqttDiscoveryPrefix := MqttDiscoveryPrefix;
THIS^.MqttDiagnosticTopic := MqttDiagnosticTopic;
THIS^.pMqttPublishQueue := pMqttPublishQueue; 
                
END_METHOD
END_FUNCTION_BLOCK

{attribute 'reflection'}
FUNCTION_BLOCK FB_BASE_MQTT_DISCOVERY_DEVICE
  VAR
    name : STRING;
    cu : STRING;  (* configuration_url *)
    ids : STRING;  (* identifiers *)
    mf : STRING;  (* manufacturer *)
    mdl : STRING;  (* model *)
    sw : STRING;  (* sw_version *)
    hw : STRING;  (* hw_version *)
    ip : STRING;  (* Held for SendDeviceUpdate's change detection, NOT published. Home Assistant carries these in the device's "connections" field, which is a list of pairs ([["mac","aa:bb:.."]]); MQTT_DISCOVERY_DEVICE is one JSONVAR per field and cannot express a nested array, the same limitation that stops the fan platform advertising preset_modes. Publishing them needs that struct to gain real list support first. *)
    sMac : STRING;
    bInit : BOOL := TRUE;
    {attribute 'noinit'}
    {attribute 'instance-path'}
    sInstanceName : STRING(GVL_MQTT.MQTT_TOPIC_LEN);  (* object's full instance name *)
    pMqttPublishQueue : POINTER TO FB_MQTT_PUBLISH_QUEUE;
    availabilityTopic1 : STRING(GVL_MQTT.MQTT_TOPIC_LEN);
    availabilityTopic2 : STRING(GVL_MQTT.MQTT_TOPIC_LEN);
    availabilityOnline : STRING;
    availabilityOffline : STRING;
    MqttDiscoveryPrefix : STRING;
    MqttDiagnosticTopic : STRING(GVL_MQTT.MQTT_TOPIC_LEN);
    stMqttDiscMsgBinSens : MQTT_DISCOVERY_BINARY_SENSOR;
    stMqttDiscMsgBinSensWCat : MQTT_DISCOVERY_BINARY_SENSOR_ENT_CAT;
    stMqttDiscMsgCover : MQTT_DISCOVERY_COVER;
    stMqttDiscMsgLightDim : MQTT_DISCOVERY_LIGHT_DIMMER;
    stMqttDiscMsgLight : MQTT_DISCOVERY_LIGHT;
    stMqttDiscMsgLock : MQTT_DISCOVERY_LOCK;
    stMqttDiscMsgSensor : MQTT_DISCOVERY_SENSOR;
    stMqttDiscMsgSensorDiagnostic : MQTT_DISCOVERY_SENSOR_DIAGNOSTIC;
    stMqttDiscMsgSiren : MQTT_DISCOVERY_SIREN;
    stMqttDiscMsgSwitch : MQTT_DISCOVERY_SWITCH;
    stMqttDiscMsgClimate : MQTT_DISCOVERY_CLIMATE;
    stMqttDiscMsgEvent : MQTT_DISCOVERY_EVENT;
    stMqttDiscMsgValveState : MQTT_DISCOVERY_VALVE_STATE;
    stMqttDiscMsgValve : MQTT_DISCOVERY_VALVE;
    stMqttDiscMsgFan : MQTT_DISCOVERY_FAN;  (* Home Assistant fan platform *)
    stMqttDiscMsgCoverPos : MQTT_DISCOVERY_COVER_POSITION;  (* The position-capable cover's own config struct. A separate struct because Home Assistant rejects position_topic and set_position_topic as null, so a cover without a slider has to publish a config where those keys are absent rather than empty - see CreateCoverEntityWithPosition. *)
    stMqttDiscMsgNumber : MQTT_DISCOVERY_NUMBER;  (* One instance per entity kind, reused across every announcement. The config is composed and published inside the Create* method, so nothing here has to outlive the call - which is why sixteen of these cost one struct each rather than one per entity. *)
    stMqttDiscMsgButton : MQTT_DISCOVERY_BUTTON;
    iQueueLane : INT := 0;  (* Which publish-queue lane this device's messages go on. A lane must have exactly one producing task, and this object is used from several - the owner sets it, defaulting to the same lane everything else uses. *)
  END_VAR

            
          

METHOD CreateDiagnosticSensorEntity
  VAR_INPUT
    Name : STRING;  (* default *)
    Id : STRING;
    StateTopic : STRING(GVL_MQTT.MQTT_TOPIC_LEN);  (* entity specific *)
    StateValue : STRING := '';
    ExpiryAfter : INT := 0;
    UnitOfMeasurement : STRING := '';
    StateClass : STRING := '';
  END_VAR
  VAR
    EntityId : STRING(25) := 'sensor';
  END_VAR
                  (* Name, id, availability and device are identical for every entity type, so
   they are filled once through the shared base struct. *)
THIS^.FillCommonFields(
	pBase := ADR(stMqttDiscMsgSensorDiagnostic),
	EntityId := EntityId,
	Name := name,
	Id := Id);

// Entity related: Specific
//MqttDiscoverySensorMessage.ic.CharString := Icon;
stMqttDiscMsgSensorDiagnostic.stat_t.CharString := StateTopic;
stMqttDiscMsgSensorDiagnostic.exp_aft.Integer := ExpiryAfter;
stMqttDiscMsgSensorDiagnostic.ent_cat.CharString := 'diagnostic';

(* Optional, and left out of the JSON entirely when not given, so every existing
   diagnostic entity is unaffected. *)
IF NOT CommonTypesAndFunctions.StrEquals(str1 := ADR(UnitOfMeasurement), str2 := ADR('')) THEN
	stMqttDiscMsgSensorDiagnostic.unit_of_meas.CharString := UnitOfMeasurement;
END_IF
IF NOT CommonTypesAndFunctions.StrEquals(str1 := ADR(StateClass), str2 := ADR('')) THEN
	stMqttDiscMsgSensorDiagnostic.stat_cla.CharString := StateClass;
END_IF



IF THIS^.PublishEntityConfig(
		pStruct := ADR(stMqttDiscMsgSensorDiagnostic),
		StructSize := SIZEOF(stMqttDiscMsgSensorDiagnostic),
		EntityId := EntityId,
		Id := Id) AND NOT (StateValue = '') THEN
	(* This entity seeds its own initial value as well as its config. *)
	pMqttPublishQueue^.AddMessageOn(Lane := iQueueLane,
		Payload:= StateValue,
		Topic := StateTopic,
		Qos := MQTT.QoS.ExactlyOnce,
		MqttRetain := TRUE,
	);
END_IF
                
END_METHOD

